IF  Mach_Control.U.WJ_iMode=3 AND arrAxisCtrl[AxiseNo.AxisName.TailCurlLine].Status.Homed 
AND arrAxisCtrl[AxiseNo.AxisName.TailCurlWhirling].Cmd.arrbRealPoint[1] 
AND arrAxisCtrl[AxiseNo.AxisName.LCurlingneedleLine].Status.fActPos<=arrAxisPar[AxiseNo.AxisName.LCurlingneedleLine].arrTargetPoint[1] +1
AND arrAxisCtrl[AxiseNo.AxisName.LCurlingneedleLine].Status.Homed  
AND arrAxisCtrl[AxiseNo.AxisName.SCurlingneedleLine].Status.fActPos <=arrAxisPar[AxiseNo.AxisName.SCurlingneedleLine] .arrTargetPoint[1] +1
AND arrAxisCtrl[AxiseNo.AxisName.SCurlingneedleLine].Status.Homed 
OR Mach_Control.WJ_b.AxisConditionEN THEN
	arrAxisCtrl[AxiseNo.AxisName.TailCurlLine].Cmd.GoPoint_Condition[10]:=TRUE;
ELSE
	arrAxisCtrl[AxiseNo.AxisName.TailCurlLine].Cmd.GoPoint_Condition[10]:=FALSE;	
END_IF

IF  Mach_Control.U.WJ_iMode=3 AND   arrAxisCtrl[AxiseNo.AxisName.TailCurlLine].Status.Homed  AND   arrAxisCtrl[AxiseNo.AxisName.TailCurlWhirling].Cmd.arrbRealPoint[1] AND
	(arrAxisCtrl[AxiseNo.AxisName.LCurlingneedleLine].Status.fActPos<=arrAxisPar[AxiseNo.AxisName.LCurlingneedleLine].arrTargetPoint[1]+1 AND arrAxisCtrl[AxiseNo.AxisName.LCurlingneedleLine].Status.Homed  AND
	arrAxisCtrl[AxiseNo.AxisName.SCurlingneedleLine].Status.fActPos <=arrAxisPar[AxiseNo.AxisName.SCurlingneedleLine] .arrTargetPoint[1]+1 AND arrAxisCtrl[AxiseNo.AxisName.SCurlingneedleLine].Status.Homed  AND
	arrAxisCtrl[AxiseNo.AxisName.TailCurlSEPTAUpDown].Cmd.arrbRealPoint[1] ) AND  arrCyCtrl[arrCyNo.CylinderName.PoleSplintCy_D].Status.OFFState AND
    arrAxisCtrl[AxiseNo.AxisName.TailCurlSEPTALine].Cmd.arrbRealPoint[1] OR Mach_Control.WJ_b.AxisConditionEN THEN
    arrAxisCtrl[AxiseNo.AxisName.TailCurlLine].Cmd.GoPoint_Condition[11]:=TRUE;
ELSE
	arrAxisCtrl[AxiseNo.AxisName.TailCurlLine].Cmd.GoPoint_Condition[11]:=FALSE;	
END_IF


//尾卷夹电芯伸缩
IF  Mach_Control.U.WJ_iMode=3  
OR Mach_Control.WJ_b.AxisConditionEN THEN
	arrAxisCtrl[AxiseNo.AxisName.TailCurlRetracting].Cmd.Home_Condition:=TRUE;
ELSE
	arrAxisCtrl[AxiseNo.AxisName.TailCurlRetracting].Cmd.Home_Condition:=FALSE;	
END_IF

IF  Mach_Control.U.WJ_iMode=3 AND arrAxisCtrl[AxiseNo.AxisName.TailCurlRetracting].Status.Homed 
OR Mach_Control.WJ_b.AxisConditionEN THEN
	arrAxisCtrl[AxiseNo.AxisName.TailCurlRetracting].Cmd.GoPoint_Condition[1]:=TRUE;
ELSE
	arrAxisCtrl[AxiseNo.AxisName.TailCurlRetracting].Cmd.GoPoint_Condition[1]:=FALSE;	
END_IF

IF  Mach_Control.U.WJ_iMode=3 AND arrAxisCtrl[AxiseNo.AxisName.TailCurlRetracting].Status.Homed 
OR Mach_Control.WJ_b.AxisConditionEN THEN
	arrAxisCtrl[AxiseNo.AxisName.TailCurlRetracting].Cmd.GoPoint_Condition[2]:=TRUE;
ELSE
	arrAxisCtrl[AxiseNo.AxisName.TailCurlRetracting].Cmd.GoPoint_Condition[2]:=FALSE;	
END_IF

IF  Mach_Control.U.WJ_iMode=3 AND arrAxisCtrl[AxiseNo.AxisName.TailCurlRetracting].Status.Homed 
OR Mach_Control.WJ_b.AxisConditionEN THEN
	arrAxisCtrl[AxiseNo.AxisName.TailCurlRetracting].Cmd.GoPoint_Condition[3]:=TRUE;
ELSE
	arrAxisCtrl[AxiseNo.AxisName.TailCurlRetracting].Cmd.GoPoint_Condition[3]:=FALSE;	
END_IF


//尾卷夹膜平移
IF  Mach_Control.U.WJ_iMode=3 AND
    arrAxisCtrl[AxiseNo.AxisName.CaDTCarryingUpDown].Status.fActPos<=arrAxisPar[AxiseNo.AxisName.CaDTCarryingUpDown].arrTargetPoint[5]+1 AND arrAxisCtrl[AxiseNo.AxisName.CaDTCarryingUpDown].Status.Homed AND
	arrAxisCtrl[AxiseNo.AxisName.CaDTCarryingLine].Status.Homed AND arrAxisCtrl[AxiseNo.AxisName.CaDTCarryingLine].Cmd.arrbRealPoint[1] 	 THEN
       arrAxisCtrl[AxiseNo.AxisName.TailCurlSEPTALine].Cmd.JogP_Condition:=TRUE;
ELSE 
	   arrAxisCtrl[AxiseNo.AxisName.TailCurlSEPTALine].Cmd.JogP_Condition:=FALSE;
END_IF 
 
IF  Mach_Control.U.WJ_iMode=3 AND
	arrAxisCtrl[AxiseNo.AxisName.TailCurlLine].Status.fActPos<=arrAxisPar[AxiseNo.AxisName.TailCurlLine].arrTargetPoint[4]+1 AND arrAxisCtrl[AxiseNo.AxisName.TailCurlLine].Status.Homed 
    OR Mach_Control.WJ_b.AxisConditionEN THEN
		arrAxisCtrl[AxiseNo.AxisName.TailCurlSEPTALine].Cmd.Home_Condition:=TRUE;
		arrAxisCtrl[AxiseNo.AxisName.TailCurlSEPTALine].Cmd.GoPoint_Condition[1]:=TRUE;
		//TailCurlSEPTALineGoargee:=TRUE;
ELSE
		arrAxisCtrl[AxiseNo.AxisName.TailCurlSEPTALine].Cmd.Home_Condition:=FALSE;	
		arrAxisCtrl[AxiseNo.AxisName.TailCurlSEPTALine].Cmd.GoPoint_Condition[1]:=FALSE;
		//TailCurlSEPTALineGoargee:=FALSE;
END_IF

IF  Mach_Control.U.WJ_iMode=3 AND
	arrAxisCtrl[AxiseNo.AxisName.CaDTCarryingUpDown].Status.fActPos<=arrAxisPar[AxiseNo.AxisName.CaDTCarryingUpDown].arrTargetPoint[5]+1 AND arrAxisCtrl[AxiseNo.AxisName.CaDTCarryingUpDown].Status.Homed AND
	arrAxisCtrl[AxiseNo.AxisName.CaDTCarryingLine].Status.Homed AND arrAxisCtrl[AxiseNo.AxisName.CaDTCarryingLine].Cmd.arrbRealPoint[1] 
OR Mach_Control.WJ_b.AxisConditionEN THEN
		arrAxisCtrl[AxiseNo.AxisName.TailCurlSEPTALine].Cmd.Home_Condition:=TRUE;

		arrAxisCtrl[AxiseNo.AxisName.TailCurlSEPTALine].Cmd.GoPoint_Condition[2]:=TRUE;
		//TailCurlSEPTALineGoargee:=TRUE;
ELSE
		arrAxisCtrl[AxiseNo.AxisName.TailCurlSEPTALine].Cmd.Home_Condition:=FALSE;	

		arrAxisCtrl[AxiseNo.AxisName.TailCurlSEPTALine].Cmd.GoPoint_Condition[2]:=FALSE;
		//TailCurlSEPTALineGoargee:=FALSE;
END_IF

(*
IF  Mach_Control.U.DT_iMode=3 AND arrAxisCtrl[AxiseNo.AxisName.CaCarryingLine2].Cmd.arrbRealPoint[1] 
AND (arrAxisCtrl[AxiseNo.AxisName.TailCurlLine].Cmd.arrbRealPoint[5] OR arrAxisCtrl[AxiseNo.AxisName.TailCurlLine].Cmd.arrbRealPoint[6] OR arrAxisCtrl[AxiseNo.AxisName.TailCurlLine].Cmd.arrbRealPoint[1])
AND (arrAxisCtrl[AxiseNo.AxisName.TailCurlWhirling].Cmd.arrbRealPoint[1] OR  arrAxisCtrl[AxiseNo.AxisName.TailCurlWhirling].Cmd.arrbRealPoint[2]) THEN
	arrAxisCtrl[AxiseNo.AxisName.TailCurlSEPTALine].Cmd.GoPoint_Condition[1]:=TRUE;
ELSE
	arrAxisCtrl[AxiseNo.AxisName.TailCurlSEPTALine].Cmd.GoPoint_Condition[1]:=FALSE;	
END_IF

IF  Mach_Control.U.DT_iMode=3 AND arrAxisCtrl[AxiseNo.AxisName.CaCarryingLine2].Cmd.arrbRealPoint[1] 
AND (arrAxisCtrl[AxiseNo.AxisName.TailCurlLine].Cmd.arrbRealPoint[5] OR arrAxisCtrl[AxiseNo.AxisName.TailCurlLine].Cmd.arrbRealPoint[6] OR arrAxisCtrl[AxiseNo.AxisName.TailCurlLine].Cmd.arrbRealPoint[1])
AND (arrAxisCtrl[AxiseNo.AxisName.TailCurlWhirling].Cmd.arrbRealPoint[1] OR  arrAxisCtrl[AxiseNo.AxisName.TailCurlWhirling].Cmd.arrbRealPoint[2]) THEN
	arrAxisCtrl[AxiseNo.AxisName.TailCurlSEPTALine].Cmd.GoPoint_Condition[2]:=TRUE;
ELSE
	arrAxisCtrl[AxiseNo.AxisName.TailCurlSEPTALine].Cmd.GoPoint_Condition[2]:=FALSE;	
END_IF
*)

//尾卷夹膜升降
IF  Mach_Control.U.WJ_iMode=3 AND
	 arrAxisCtrl[AxiseNo.AxisName.TailCurlLine].Status.fSetPos<=arrAxisPar[AxiseNo.AxisName.TailCurlLine].arrTargetPoint[4] AND arrAxisCtrl[AxiseNo.AxisName.TailCurlLine].Status.Homed    
OR Mach_Control.WJ_b.AxisConditionEN THEN
		arrAxisCtrl[AxiseNo.AxisName.TailCurlSEPTAUpDown].Cmd.Home_Condition:=TRUE;
ELSE
	arrAxisCtrl[AxiseNo.AxisName.TailCurlSEPTAUpDown].Cmd.Home_Condition:=FALSE;	
END_IF

IF  Mach_Control.U.WJ_iMode=3 AND arrAxisCtrl[AxiseNo.AxisName.TailCurlSEPTAUpDown].Status.Homed 
AND NOT arrAxisCtrl[AxiseNo.AxisName.TailCurlLine].Cmd.arrbRealPoint[11] OR Mach_Control.WJ_b.AxisConditionEN THEN
	arrAxisCtrl[AxiseNo.AxisName.TailCurlSEPTAUpDown].Cmd.GoPoint_Condition[1]:=TRUE;
ELSE
	arrAxisCtrl[AxiseNo.AxisName.TailCurlSEPTAUpDown].Cmd.GoPoint_Condition[1]:=FALSE;	
END_IF

IF  Mach_Control.U.WJ_iMode=3 AND arrAxisCtrl[AxiseNo.AxisName.TailCurlSEPTAUpDown].Status.Homed  
AND arrAxisCtrl[AxiseNo.AxisName.TailCurlLine].Status.fActPos <=  arrAxisPar[AxiseNo.AxisName.TailCurlLine].arrTargetPoint[4]  
AND NOT arrAxisCtrl[AxiseNo.AxisName.TailCurlLine].Cmd.arrbRealPoint[11] OR Mach_Control.WJ_b.AxisConditionEN THEN
	arrAxisCtrl[AxiseNo.AxisName.TailCurlSEPTAUpDown].Cmd.GoPoint_Condition[2]:=TRUE;
ELSE
	arrAxisCtrl[AxiseNo.AxisName.TailCurlSEPTAUpDown].Cmd.GoPoint_Condition[2]:=FALSE;	
END_IF

//尾卷夹电芯升降
IF  Mach_Control.U.WJ_iMode=3 AND  arrAxisCtrl[AxiseNo.AxisName.TailCurlRetracting].Cmd.arrbRealPoint[1] 
OR Mach_Control.WJ_b.AxisConditionEN THEN
	arrAxisCtrl[AxiseNo.AxisName.TailCurlUpDown].Cmd.Home_Condition:=TRUE;
ELSE
	arrAxisCtrl[AxiseNo.AxisName.TailCurlUpDown].Cmd.Home_Condition:=FALSE;	
END_IF

IF  Mach_Control.U.WJ_iMode=3 
AND arrAxisCtrl[AxiseNo.AxisName.TailCurlSEPTAUpDown].Status.Homed  
AND  arrAxisCtrl[AxiseNo.AxisName.TailCurlRetracting].Cmd.arrbRealPoint[1] 
AND NOT arrAxisCtrl[AxiseNo.AxisName.TailCurlLine].Cmd.arrbRealPoint[6]
OR Mach_Control.WJ_b.AxisConditionEN THEN
	arrAxisCtrl[AxiseNo.AxisName.TailCurlUpDown].Cmd.GoPoint_Condition[1]:=TRUE;
ELSE
	arrAxisCtrl[AxiseNo.AxisName.TailCurlUpDown].Cmd.GoPoint_Condition[1]:=FALSE;	
END_IF
////////////////////////////////////////////
IF  Mach_Control.U.WJ_iMode=3 
AND arrAxisCtrl[AxiseNo.AxisName.TailCurlSEPTAUpDown].Status.Homed  
AND arrAxisCtrl[AxiseNo.AxisName.TailCurlWhirling].Cmd.arrbRealPoint[1]
AND arrAxisCtrl[AxiseNo.AxisName.TailCurlRetracting].Cmd.arrbRealPoint[1] 
AND  arrAxisCtrl[AxiseNo.AxisName.TailCurlLine].Status.fActPos <=  arrAxisPar[AxiseNo.AxisName.TailCurlLine].arrTargetPoint[4]  
OR Mach_Control.WJ_b.AxisConditionEN THEN
	arrAxisCtrl[AxiseNo.AxisName.TailCurlUpDown].Cmd.GoPoint_Condition[2]:=TRUE;
ELSE
	arrAxisCtrl[AxiseNo.AxisName.TailCurlUpDown].Cmd.GoPoint_Condition[2]:=FALSE;	
END_IF

IF  Mach_Control.U.WJ_iMode=3 
AND arrAxisCtrl[AxiseNo.AxisName.TailCurlSEPTAUpDown].Status.Homed 
AND arrAxisCtrl[AxiseNo.AxisName.TailCurlRetracting].Cmd.arrbRealPoint[1]
AND NOT arrAxisCtrl[AxiseNo.AxisName.TailCurlLine].Cmd.arrbRealPoint[11] 
OR Mach_Control.WJ_b.AxisConditionEN THEN
	arrAxisCtrl[AxiseNo.AxisName.TailCurlUpDown].Cmd.GoPoint_Condition[3]:=TRUE;

ELSE
	arrAxisCtrl[AxiseNo.AxisName.TailCurlUpDown].Cmd.GoPoint_Condition[3]:=FALSE;	
END_IF

IF  Mach_Control.U.WJ_iMode=3 
AND arrAxisCtrl[AxiseNo.AxisName.TailCurlSEPTAUpDown].Status.Homed
AND arrAxisCtrl[AxiseNo.AxisName.TailCurlWhirling].Cmd.arrbRealPoint[2]  
AND arrAxisCtrl[AxiseNo.AxisName.TailCurlRetracting].Cmd.arrbRealPoint[1]
AND NOT arrAxisCtrl[AxiseNo.AxisName.TailCurlLine].Cmd.arrbRealPoint[11] 
OR Mach_Control.WJ_b.AxisConditionEN THEN
	arrAxisCtrl[AxiseNo.AxisName.TailCurlUpDown].Cmd.GoPoint_Condition[4]:=TRUE;
ELSE
	arrAxisCtrl[AxiseNo.AxisName.TailCurlUpDown].Cmd.GoPoint_Condition[4]:=FALSE;	
END_IF
///////////////////////////////////////////
//尾卷夹电芯旋转 
IF  Mach_Control.U.WJ_iMode=3 AND  arrAxisCtrl[AxiseNo.AxisName.TailCurlRetracting].Cmd.arrbRealPoint[1] AND arrAxisCtrl[AxiseNo.AxisName.TailCurlLine].Cmd.arrbRealPoint[1] AND
   arrAxisCtrl[AxiseNo.AxisName.TailCurlRetracting].Status.Homed AND arrAxisCtrl[AxiseNo.AxisName.TailCurlLine].Status.Homed 	
OR Mach_Control.WJ_b.AxisConditionEN THEN
	arrAxisCtrl[AxiseNo.AxisName.TailCurlWhirling].Cmd.Home_Condition:=TRUE;
ELSE
	arrAxisCtrl[AxiseNo.AxisName.TailCurlWhirling].Cmd.Home_Condition:=FALSE;	
END_IF

IF  Mach_Control.U.WJ_iMode=3 AND arrAxis[AxiseNo.AxisName.TailCurlWhirling].Status.Homed  AND  arrAxisCtrl[AxiseNo.AxisName.TailCurlRetracting].Cmd.arrbRealPoint[1] 
AND arrAxisCtrl[AxiseNo.AxisName.TailCurlUpDown].Cmd.arrbRealPoint[3] AND arrAxisCtrl[AxiseNo.AxisName.TailCurlLine].Cmd.arrbRealPoint[1] 
OR Mach_Control.WJ_b.AxisConditionEN THEN
	arrAxisCtrl[AxiseNo.AxisName.TailCurlWhirling].Cmd.GoPoint_Condition[1]:=TRUE;
ELSE
	arrAxisCtrl[AxiseNo.AxisName.TailCurlWhirling].Cmd.GoPoint_Condition[1]:=FALSE;	
END_IF

IF  Mach_Control.U.WJ_iMode=3 AND arrAxis[AxiseNo.AxisName.TailCurlWhirling].Status.Homed  AND  arrAxisCtrl[AxiseNo.AxisName.TailCurlRetracting].Cmd.arrbRealPoint[1] 
AND arrAxisCtrl[AxiseNo.AxisName.TailCurlUpDown].Cmd.arrbRealPoint[3] AND arrAxisCtrl[AxiseNo.AxisName.TailCurlLine].Cmd.arrbRealPoint[1] 
OR Mach_Control.WJ_b.AxisConditionEN THEN
	arrAxisCtrl[AxiseNo.AxisName.TailCurlWhirling].Cmd.GoPoint_Condition[2]:=TRUE;
ELSE
	arrAxisCtrl[AxiseNo.AxisName.TailCurlWhirling].Cmd.GoPoint_Condition[2]:=FALSE;	
END_IF

//尾卷长卷针平移
IF  Mach_Control.U.WJ_iMode=3 
OR Mach_Control.WJ_b.AxisConditionEN THEN
	arrAxisCtrl[AxiseNo.AxisName.LCurlingneedleLine].Cmd.Home_Condition:=TRUE;
ELSE
	arrAxisCtrl[AxiseNo.AxisName.LCurlingneedleLine].Cmd.Home_Condition:=FALSE;	
END_IF

IF  Mach_Control.U.WJ_iMode=3 AND arrAxisCtrl[AxiseNo.AxisName.LCurlingneedleLine].Status.Homed AND arrCyCtrl[arrCyNo.CylinderName.CurlingSplintCy_L].Status.OFFState
OR Mach_Control.WJ_b.AxisConditionEN THEN
	arrAxisCtrl[AxiseNo.AxisName.LCurlingneedleLine].Cmd.GoPoint_Condition[1]:=TRUE;
ELSE
	arrAxisCtrl[AxiseNo.AxisName.LCurlingneedleLine].Cmd.GoPoint_Condition[1]:=FALSE;	
END_IF

IF  Mach_Control.U.WJ_iMode=3 AND arrAxisCtrl[AxiseNo.AxisName.LCurlingneedleLine].Status.Homed AND arrCyCtrl[arrCyNo.CylinderName.CurlingSplintCy_L].Status.OFFState
     AND  arrAxisCtrl[AxiseNo.AxisName.TailCurlLine].Cmd.arrbRealPoint[4]   OR Mach_Control.WJ_b.AxisConditionEN THEN
	arrAxisCtrl[AxiseNo.AxisName.LCurlingneedleLine].Cmd.GoPoint_Condition[2]:=TRUE;
ELSE
	arrAxisCtrl[AxiseNo.AxisName.LCurlingneedleLine].Cmd.GoPoint_Condition[2]:=FALSE;	
END_IF


//尾卷短卷针平移
IF  (Mach_Control.U.WJ_iMode=3  AND arrAxisCtrl[AxiseNo.AxisName.SCurlingneedleWhirling].Io.biHomeSwitch)
OR Mach_Control.WJ_b.AxisConditionEN   THEN
	arrAxisCtrl[AxiseNo.AxisName.SCurlingneedleLine].Cmd.Home_Condition:=TRUE;
ELSE
	arrAxisCtrl[AxiseNo.AxisName.SCurlingneedleLine].Cmd.Home_Condition:=FALSE;	
END_IF

IF  Mach_Control.U.WJ_iMode=3 AND arrAxisCtrl[AxiseNo.AxisName.SCurlingneedleLine].Status.Homed  AND arrCyCtrl[arrCyNo.CylinderName.CurlingSplintCy_S].Status.OFFState
OR Mach_Control.WJ_b.AxisConditionEN THEN
	arrAxisCtrl[AxiseNo.AxisName.SCurlingneedleLine].Cmd.GoPoint_Condition[1]:=TRUE;
ELSE
	arrAxisCtrl[AxiseNo.AxisName.SCurlingneedleLine].Cmd.GoPoint_Condition[1]:=FALSE;	
END_IF

IF  Mach_Control.U.WJ_iMode=3 AND arrAxisCtrl[AxiseNo.AxisName.SCurlingneedleLine].Status.Homed  AND arrCyCtrl[arrCyNo.CylinderName.CurlingSplintCy_S].Status.OFFState
    AND  arrCyCtrl[arrCyNo.ElectValveName.WJShortvacuum].Io.DOStatus1 AND  arrAxisCtrl[AxiseNo.AxisName.TailCurlLine].Cmd.arrbRealPoint[4]    OR Mach_Control.WJ_b.AxisConditionEN THEN
	arrAxisCtrl[AxiseNo.AxisName.SCurlingneedleLine].Cmd.GoPoint_Condition[2]:=TRUE;
ELSE
	arrAxisCtrl[AxiseNo.AxisName.SCurlingneedleLine].Cmd.GoPoint_Condition[2]:=FALSE;	
END_IF

//尾卷长卷针旋转
IF  Mach_Control.U.WJ_iMode=3 AND arrAxisCtrl[AxiseNo.AxisName.LCurlingneedleLine].Status.fSetPos<=arrAxisPar[AxiseNo.AxisName.LCurlingneedleLine].arrTargetPoint[1]  
OR Mach_Control.WJ_b.AxisConditionEN THEN
	arrAxisCtrl[AxiseNo.AxisName.LCurlingneedleWhirling].Cmd.Home_Condition:=TRUE;
ELSE
	arrAxisCtrl[AxiseNo.AxisName.LCurlingneedleWhirling].Cmd.Home_Condition:=FALSE;	
END_IF

IF  Mach_Control.U.WJ_iMode=3 AND arrAxisCtrl[AxiseNo.AxisName.LCurlingneedleWhirling].Status.Homed 
AND arrAxisCtrl[AxiseNo.AxisName.LCurlingneedleLine].Cmd.arrbRealPoint[1]  
OR Mach_Control.WJ_b.AxisConditionEN THEN
	arrAxisCtrl[AxiseNo.AxisName.LCurlingneedleWhirling].Cmd.GoPoint_Condition[1]:=TRUE;
ELSE
	arrAxisCtrl[AxiseNo.AxisName.LCurlingneedleWhirling].Cmd.GoPoint_Condition[1]:=FALSE;	
END_IF

//尾卷短卷针旋转
IF  Mach_Control.U.WJ_iMode=3 AND arrAxisCtrl[AxiseNo.AxisName.SCurlingneedleLine].Status.fSetPos<=arrAxisPar[AxiseNo.AxisName.SCurlingneedleLine].arrTargetPoint[1]  
OR Mach_Control.WJ_b.AxisConditionEN THEN
	arrAxisCtrl[AxiseNo.AxisName.SCurlingneedleWhirling].Cmd.Home_Condition:=TRUE;
ELSE
	arrAxisCtrl[AxiseNo.AxisName.SCurlingneedleWhirling].Cmd.Home_Condition:=FALSE;	
END_IF

IF  Mach_Control.U.WJ_iMode=3 AND arrAxisCtrl[AxiseNo.AxisName.SCurlingneedleWhirling].Status.Homed 
AND arrAxisCtrl[AxiseNo.AxisName.SCurlingneedleLine].Cmd.arrbRealPoint[1]  
OR Mach_Control.WJ_b.AxisConditionEN THEN
	arrAxisCtrl[AxiseNo.AxisName.SCurlingneedleWhirling].Cmd.GoPoint_Condition[1]:=TRUE;
ELSE
	arrAxisCtrl[AxiseNo.AxisName.SCurlingneedleWhirling].Cmd.GoPoint_Condition[1]:=FALSE;	
END_IF
END_ACTION

ACTION TailCurl_Gohome:
Tailcurl_GohomeOverTon(IN:= , PT:=T#90S , Q=> , ET=> );//叠台回原点超时报警延时

//判断回原点的状态
IF arrAxisCtrl[AxiseNo.AxisName.SCurlingneedleLine].Status.Homed AND arrAxisCtrl[AxiseNo.AxisName.LCurlingneedleLine].Status.Homed AND 
	arrAxisCtrl[AxiseNo.AxisName.LCurlingneedleWhirling].Status.Homed  AND arrAxisCtrl[AxiseNo.AxisName.SCurlingneedleWhirling].Status.Homed AND 
	arrAxisCtrl[AxiseNo.AxisName.TailCurlLine].Status.Homed AND arrAxisCtrl[AxiseNo.AxisName.TailCurlRetracting].Status.Homed AND 
	arrAxisCtrl[AxiseNo.AxisName.TailCurlUpDown].Status.Homed AND arrAxisCtrl[AxiseNo.AxisName.TailCurlSEPTAUpDown].Status.Homed AND 
	arrAxis[AxiseNo.AxisName.TailCurlSEPTALine].Status.Homed AND arrAxis[AxiseNo.AxisName.TailCurlWhirling].Status.Homed AND WZIniti_Done THEN
		Mach_Control.WJ_b.WZIniti_Done:=TRUE;//初始化完成	
ELSE
		Mach_Control.WJ_b.WZIniti_Done:=FALSE;//初始化完成	
END_IF

IF Mach_Control.U.WJ_iMode=3 THEN//在手动状态下
	IF  Tailcurl_Gohoming THEN
			IF 	NOT Tailcurl_GohomeOverTon.Q THEN
				    Tailcurl_GohomeOverTon.IN:=TRUE;
			ELSE
				IF 	Tailcurl_GohomeOverTon.Q THEN
					Tailcurl_Gohoming:=FALSE;
					TailCurlStep1:=0;
				     Mach_Control.WJ_b.Error[19]:=TRUE;//尾卷回原点超时报警
				     Tailcurl_GohomeOverTon.IN:=FALSE;
				END_IF	 
					 
			END_IF
	
	ELSE
			Tailcurl_GohomeOverTon.IN:=FALSE;
	END_IF
	
	IF r_TailCurl_init.Q THEN
		Tailcurl_GohomeDone:=FALSE;//尾卷回原点完成
		Tailcurl_Gohoming:=FALSE;//尾卷回原点中
		TailCurlStep1:=0;
		Mach_Control.WJ_b.WZIniti_Done:=FALSE;//负极取片回原点完成
		WZIniti_Done:=FALSE;//负极取片回原点完成
	END_IF	

	//尾卷贴胶初始化
	r_TailCurl_init(CLK:=Mach_Control.WJ_b.WZIniti_Hbtn , Q=> );
	f_TailCurl_init(CLK:=Mach_Control.WJ_b.WZIniti_Hbtn   , Q=> );
	tTailCurlTON(IN:= , PT:=T#0.5S , Q=> , ET=> );
	CASE TailCurlStep1 OF
	0://启动尾卷贴胶初始化，气缸复位
		IF f_TailCurl_init.Q THEN	
			Tailcurl_GohomeDone:=FALSE;//尾卷回原点完成
		    Tailcurl_Gohoming:=TRUE;//尾卷回原点中
			TailCurlStep1:=1;
		END_IF
	1://回原点完成复位
			WZIniti_Done:=FALSE;//初始化完成	
			TailCurlStep3 :=0;
			TailCurlStep4:=0;
			TailCurlStep5:=0;
			TailCurlStep6:=0;
			
			arrAxisCtrl[AxiseNo.AxisName.TailCurlSEPTALine].Cmd.fOverride:=100;
			arrAxisCtrl[AxiseNo.AxisName.TailCurlRetracting].Cmd.fOverride:=100;
			arrAxisCtrl[AxiseNo.AxisName.TailCurlLine].Cmd.fOverride:=100;
						
			tailCult_GearInMultiMaster.Enable:=FALSE;
			tailCurlGearInEnable:=FALSE;
			tailCurlGearInEnable1:=FALSE;
			tailRetGearInEnable:=FALSE;//夹电芯平移与夹电芯伸缩电子齿轮
			CurlingneedleLineEnable:=FALSE;
			tailCult_GearInMultiMaster.Enable:=FALSE;
			
			 Mach_Control.DT_b.OffloadDone:=FALSE;
			 Mach_Control.WJ_b.TailCurlDone	:=FALSE;
			 //Mach_Control.DT_b.OffloadRequest:=FALSE;//复位电芯下料请求	
			 Mach_Control.WJ_b.TailCultOffloading:=FALSE;
			CellMemory[Mach_Control.WJ_b.WJ_Memory].Cell:=FALSE;	
			TailCurlStart:=FALSE;//复位尾卷启动
			Mach_Control.WJ_b.TailCurlDone	:=FALSE;	//尾卷完成
			arrAxisCtrl[AxiseNo.VirAxisName.VirTailCurl].Cmd.bMoveAbs:=FALSE;//主轴启动
			CurlingneedleLineEnable:=FALSE;//长、短卷针平移电子齿轮耦合启动
			tailCurlGearInEnable:=FALSE;//电子齿轮耦合		
			tTailCurlTON.IN:=FALSE;
			arrAxisCtrl[AxiseNo.AxisName.TailCurlSEPTALine].Cmd.bDynamitcsParSel:=1;
			fbCamInEndWindX.bGearOutMode:=FALSE;//夹膜平移轴凸轮耦合
			IF NOT WZIniti_Done AND arrAxisCtrl[AxiseNo.AxisName.TailCurlSEPTALine].Cmd.bDynamitcsParSel=1 THEN
				TailCurlStep1:=10;
			END_IF
	10://气缸复位，尾卷状态复位
			IF  NOT 	tTailCurlTON.Q THEN	
					tTailCurlTON.IN:=TRUE;
					//arrCyCtrl[arrCyNo.CylinderName.CurlingSplintCy_S_1].Cmd.bON:=TRUE;//尾卷短卷针泄压关闭
					arrCyCtrl[arrCyNo.CylinderName.CurlingSplintCy_L].Cmd.bOFF:=TRUE;//尾卷长卷针张开
					arrCyCtrl[arrCyNo.CylinderName.CurlingSplintCy_S].Cmd.bOFF:=TRUE;//尾卷短卷针张开	
					arrCyCtrl[arrCyNo.ElectValveName.WJShortvacuum].Cmd.bON:=TRUE;//短卷针张开真空开
					arrCyCtrl[arrCyNo.CylinderName.PoleHotCutterCy].Cmd.bOFF:=TRUE;//隔膜热切升降气缸收回
					arrCyCtrl[arrCyNo.CylinderName.PoleSplintCy_D].Cmd.bOFF:=TRUE;//隔膜隔膜下夹板气缸收回
					arrCyCtrl[arrCyNo.CylinderName.TailCurlUpdownCy].Cmd.bOFF:=TRUE;//尾卷压轮升降气缸收回
					arrCyCtrl[arrCyNo.CylinderName.TailCurlSplintCy].Cmd.bOFF:=TRUE;//尾卷取料夹爪气缸张开	
			ELSE
					IF arrCyCtrl[arrCyNo.CylinderName.PoleHotCutterCy].Io.DIOFFSwitch AND arrCyCtrl[arrCyNo.CylinderName.PoleSplintCy_D].Io.DIOFFSwitch AND 
					   arrCyCtrl[arrCyNo.CylinderName.TailCurlUpdownCy].Io.DIOFFSwitch AND arrCyCtrl[arrCyNo.CylinderName.TailCurlSplintCy].Io.DIOFFSwitch THEN
					   tTailCurlTON.IN:=FALSE;
					   TailCurlStep1:=20;
					END_IF	
			END_IF	
	20:
			fbCamInEndWindX.bCamInExecute:=FALSE;//夹膜平移凸轮耦合
			fbCamInEndWindY.bCamInExecute:=FALSE;//夹膜升降凸轮耦合
			tailCurl1_GearIn.Execute:=FALSE;//短卷针齿轮耦合
			tailCurl2_GearIn.Execute:=FALSE;//长卷针齿轮耦合
			IF NOT fbCamInEndWindX.bCamInExecute AND NOT fbCamInEndWindY.bCamInExecute AND 
				NOT tailCurl1_GearIn.Execute AND NOT tailCurl2_GearIn.Execute THEN
				TailCurlStep1:=21;
			END_IF
	21://解除凸轮耦合
			arrCyCtrl[arrCyNo.CylinderName.TailCurlLineCy].Cmd.bOFF:=TRUE;//尾卷压轮平移气缸收回
			arrAxisCtrl[AxiseNo.AxisName.SCurlingneedleWhirling].Cmd.bGearOut:=TRUE;//尾卷短卷针旋转轴解耦
			arrAxisCtrl[AxiseNo.AxisName.LCurlingneedleWhirling].Cmd.bGearOut:=TRUE;//尾卷长卷针旋转轴解耦
			arrAxisCtrl[AxiseNo.AxisName.TailCurlLine].Cmd.bGearOut:=TRUE;//尾卷夹电芯平移轴解耦
			arrAxisCtrl[AxiseNo.AxisName.TailCurlSEPTALine].Cmd.bGearOut:=TRUE;//尾卷夹膜平移轴解耦 
			arrAxisCtrl[AxiseNo.AxisName.TailCurlSEPTAUpDown].Cmd.bGearOut:=TRUE;//尾卷夹膜升降轴解耦 
			IF NOT arrAxisCtrl[AxiseNo.AxisName.SCurlingneedleWhirling].Status.Coupled AND  NOT arrAxisCtrl[AxiseNo.AxisName.LCurlingneedleWhirling].Status.Coupled AND 
				NOT arrAxisCtrl[AxiseNo.AxisName.TailCurlLine].Status.Coupled AND NOT arrAxisCtrl[AxiseNo.AxisName.TailCurlSEPTALine].Status.Coupled AND 
				NOT arrAxisCtrl[AxiseNo.AxisName.TailCurlSEPTAUpDown].Status.Coupled THEN
				TailCurlStep1:=25;
			END_IF

	 25:
		 IF NOT arrAxisCtrl[AxiseNo.AxisName.SCurlingneedleWhirling].Io.biHomeSwitch  THEN
			  Mach_Control.WJ_b.Error[20]:=TRUE;//尾卷短卷针神伸缩回原点时,短卷针旋转原点传感器未亮报警
			  TailCurlStep1:=0;
		  ELSE 	 
			 TailCurlStep1:=30;
		 END_IF			
			

    30://尾卷长卷针伸缩轴回原点、尾卷短卷针伸缩轴回原点	
						IF NOT tTailCurlTON.Q THEN
								arrAxisCtrl[AxiseNo.AxisName.SCurlingneedleLine].Cmd.bHome:=TRUE;//尾卷短卷针平移回原点
								arrAxisCtrl[AxiseNo.AxisName.LCurlingneedleLine].Cmd.bHome:=TRUE;//尾卷长卷针平移回原点
								tTailCurlTON.IN:=TRUE;
						ELSE
								IF arrAxisCtrl[AxiseNo.AxisName.SCurlingneedleLine].Status.Homed AND arrAxisCtrl[AxiseNo.AxisName.SCurlingneedleLine].Status.NoMoving  AND
									 arrAxisCtrl[AxiseNo.AxisName.LCurlingneedleLine].Status.Homed AND arrAxisCtrl[AxiseNo.AxisName.LCurlingneedleLine].Status.NoMoving THEN
										arrAxisCtrl[AxiseNo.AxisName.SCurlingneedleLine].Cmd.bHome:=FALSE;//尾卷短卷针平移回原点
										arrAxisCtrl[AxiseNo.AxisName.LCurlingneedleLine].Cmd.bHome:=FALSE;//尾卷长卷针平移回原点
										tTailCurlTON.IN:=FALSE;
										TailCurlStep1:=35; 
								END_IF
						END_IF
			
		35:
						IF 	arrAxisCtrl[AxiseNo.AxisName.LCurlingneedleLine].Status.Homed AND arrAxisCtrl[AxiseNo.AxisName.LCurlingneedleLine].Status.NoMoving THEN
							IF arrAxisCtrl[AxiseNo.AxisName.LCurlingneedleLine].Cmd.arrbRealPoint[1] THEN
								arrAxisCtrl[AxiseNo.AxisName.LCurlingneedleLine].Cmd.iGoSetPos:=0;
							ELSE
								arrAxisCtrl[AxiseNo.AxisName.LCurlingneedleLine].Cmd.iGoSetPos:=1;//尾卷长卷针平移至初始位
							END_IF
						END_IF	
						IF 	arrAxisCtrl[AxiseNo.AxisName.SCurlingneedleLine].Status.Homed AND arrAxisCtrl[AxiseNo.AxisName.SCurlingneedleLine].Status.NoMoving THEN
							IF arrAxisCtrl[AxiseNo.AxisName.SCurlingneedleLine].Cmd.arrbRealPoint[1] THEN
								arrAxisCtrl[AxiseNo.AxisName.SCurlingneedleLine].Cmd.iGoSetPos:=0;
							ELSE
								arrAxisCtrl[AxiseNo.AxisName.SCurlingneedleLine].Cmd.iGoSetPos:=1;//尾卷短卷针平移至初始位
							END_IF
						END_IF		
							IF 	arrAxisCtrl[AxiseNo.AxisName.LCurlingneedleLine].Cmd.arrbRealPoint[1] AND arrAxisCtrl[AxiseNo.AxisName.LCurlingneedleLine].Status.NoMoving
								   AND arrAxisCtrl[AxiseNo.AxisName.SCurlingneedleLine].Cmd.arrbRealPoint[1] AND arrAxisCtrl[AxiseNo.AxisName.SCurlingneedleLine].Status.NoMoving THEN
									arrAxisCtrl[AxiseNo.AxisName.LCurlingneedleWhirling].Cmd.bHome:=FALSE;//尾卷长卷针旋转回原点
									arrAxisCtrl[AxiseNo.AxisName.SCurlingneedleWhirling].Cmd.bHome:=FALSE;//尾卷短卷针旋转回原点
									TailCurlStep1:=40; 
							END_IF
			
	40:
						IF 	arrAxisCtrl[AxiseNo.AxisName.LCurlingneedleLine].Cmd.arrbRealPoint[1] AND arrAxisCtrl[AxiseNo.AxisName.LCurlingneedleLine].Status.NoMoving AND
						arrAxisCtrl[AxiseNo.AxisName.LCurlingneedleLine].Cmd.arrbRealPoint[1] AND arrAxisCtrl[AxiseNo.AxisName.LCurlingneedleLine].Status.NoMoving THEN
						//IF NOT tTailCurlTON.Q THEN
								arrAxisCtrl[AxiseNo.AxisName.LCurlingneedleWhirling].Cmd.bHome:=TRUE;//尾卷长卷针旋转回原点
								arrAxisCtrl[AxiseNo.AxisName.SCurlingneedleWhirling].Cmd.bHome:=TRUE;//尾卷短卷针旋转回原点
								//tTailCurlTON.IN:=TRUE;
						//ELSE
								//IF arrAxisCtrl[AxiseNo.AxisName.LCurlingneedleWhirling].Status.Homed AND arrAxisCtrl[AxiseNo.AxisName.LCurlingneedleWhirling].Status.NoMoving AND 
								//	arrAxisCtrl[AxiseNo.AxisName.SCurlingneedleWhirling].Status.Homed AND arrAxisCtrl[AxiseNo.AxisName.SCurlingneedleWhirling].Status.NoMoving  THEN
									//tTailCurlTON.IN:=FALSE;
									TailCurlStep1:=50; 
								//END_IF	
						END_IF
	50://
					IF arrAxisCtrl[AxiseNo.AxisName.LCurlingneedleWhirling].Status.Homed AND arrAxisCtrl[AxiseNo.AxisName.LCurlingneedleWhirling].Status.NoMoving AND 
						arrAxisCtrl[AxiseNo.AxisName.SCurlingneedleWhirling].Status.Homed AND arrAxisCtrl[AxiseNo.AxisName.SCurlingneedleWhirling].Status.NoMoving  THEN
							TailCurlStep1:=51; 	
                            tTailCurlTON.IN:=FALSE;					
					END_IF
	51://夹电芯伸缩回原
			//IF arrAxisCtrl[AxiseNo.AxisName.TailCurlLine].Status.Homed AND arrAxisCtrl[AxiseNo.AxisName.TailCurlLine].Status.NoMoving THEN
				arrAxisCtrl[AxiseNo.AxisName.TailCurlRetracting].Cmd.bHome:=TRUE;//尾卷夹电芯伸缩回原点
				TailCurlStep1:=52; 
				tTailCurlTON.IN:=TRUE;
			//END_IF
	52:
		IF arrAxisCtrl[AxiseNo.AxisName.TailCurlRetracting].Status.Homed AND arrAxisCtrl[AxiseNo.AxisName.TailCurlRetracting].Status.NoMoving AND
           tTailCurlTON.Q  THEN
			arrAxisCtrl[AxiseNo.AxisName.TailCurlRetracting].Cmd.bHome:=FALSE;
			TailCurlStep1:=53; 
			tTailCurlTON.IN:=FALSE;
		END_IF					
					
	53://夹电芯平移回原
					IF 	arrAxisCtrl[AxiseNo.AxisName.LCurlingneedleLine].Cmd.arrbRealPoint[1] AND 	arrAxisCtrl[AxiseNo.AxisName.SCurlingneedleLine].Cmd.arrbRealPoint[1] AND 			
						arrAxisCtrl[AxiseNo.AxisName.SCurlingneedleLine].Status.Homed  AND   arrAxisCtrl[AxiseNo.AxisName.LCurlingneedleLine].Status.Homed  AND
						(arrAxisCtrl[AxiseNo.AxisName.TailCurlWhirling].Status.fSetPos<=arrAxisPar[AxiseNo.AxisName.TailCurlWhirling].arrTargetPoint[1]+1 AND
						arrAxisCtrl[AxiseNo.AxisName.TailCurlWhirling].Status.fSetPos>=arrAxisPar[AxiseNo.AxisName.TailCurlWhirling].arrTargetPoint[1]-1	) OR 
						(arrAxisCtrl[AxiseNo.AxisName.TailCurlWhirling].Status.fSetPos<=arrAxisPar[AxiseNo.AxisName.TailCurlWhirling].arrTargetPoint[2]+1 AND
						arrAxisCtrl[AxiseNo.AxisName.TailCurlWhirling].Status.fSetPos>=arrAxisPar[AxiseNo.AxisName.TailCurlWhirling].arrTargetPoint[2]-1	)  THEN
							arrAxisCtrl[AxiseNo.AxisName.TailCurlLine].Cmd.bHome:=TRUE;//尾卷夹电芯平移回原点
							TailCurlTorMark:=TRUE;//尾卷夹电芯平移力矩判断标志位
							TailCurlStep1:=54; 
							tTailCurlTON.IN:=TRUE;
                     ELSE
						    TailCurlStep1:=0; 
						     Mach_Control.WJ_b.Error[8]:=TRUE;//夹电芯平移回原点时条件不满足报警
					END_IF					
	54:
		IF arrAxisCtrl[AxiseNo.AxisName.TailCurlLine].Status.Homed AND arrAxisCtrl[AxiseNo.AxisName.TailCurlLine].Status.NoMoving AND
            tTailCurlTON.Q  THEN
			arrAxisCtrl[AxiseNo.AxisName.TailCurlLine].Cmd.bHome:=FALSE;
			TailCurlStep1:=60; 	
            tTailCurlTON.IN:=FALSE;	
		END_IF		
	
	60://夹电芯平移轴移至初始位、夹电芯伸缩轴移至初始位
						IF arrAxisCtrl[AxiseNo.AxisName.TailCurlLine].Status.Homed AND arrAxisCtrl[AxiseNo.AxisName.TailCurlLine].Status.NoMoving THEN
							TailCurlTorMark:=FALSE;//尾卷夹电芯平移力矩判断标志位
							IF arrAxisCtrl[AxiseNo.AxisName.TailCurlLine].Cmd.arrbRealPoint[1] THEN
								arrAxisCtrl[AxiseNo.AxisName.TailCurlLine].Cmd.iGoSetPos:=0;
							ELSE
								arrAxisCtrl[AxiseNo.AxisName.TailCurlLine].Cmd.iGoSetPos:=1;
							END_IF
						END_IF
						IF 	arrAxisCtrl[AxiseNo.AxisName.TailCurlRetracting].Status.Homed AND arrAxisCtrl[AxiseNo.AxisName.TailCurlRetracting].Status.NoMoving THEN
							IF arrAxisCtrl[AxiseNo.AxisName.TailCurlRetracting].Cmd.arrbRealPoint[1] THEN
								arrAxisCtrl[AxiseNo.AxisName.TailCurlRetracting].Cmd.iGoSetPos:=0;
							ELSE
								arrAxisCtrl[AxiseNo.AxisName.TailCurlRetracting].Cmd.iGoSetPos:=1;
							END_IF
						END_IF	
						IF arrAxisCtrl[AxiseNo.AxisName.TailCurlLine].Cmd.arrbRealPoint[1] AND  arrAxisCtrl[AxiseNo.AxisName.TailCurlLine].Status.NoMoving AND
							arrAxisCtrl[AxiseNo.AxisName.TailCurlRetracting].Cmd.arrbRealPoint[1] AND arrAxisCtrl[AxiseNo.AxisName.TailCurlRetracting].Status.NoMoving THEN
							TailCurlStep1:=70;
						END_IF
	70:		
			IF arrAxisCtrl[AxiseNo.AxisName.TailCurlLine].Cmd.arrbRealPoint[1] AND  arrAxisCtrl[AxiseNo.AxisName.TailCurlLine].Status.NoMoving AND
			arrAxisCtrl[AxiseNo.AxisName.TailCurlRetracting].Cmd.arrbRealPoint[1] AND arrAxisCtrl[AxiseNo.AxisName.TailCurlRetracting].Status.NoMoving THEN
			//IF NOT tTailCurlTON.Q THEN
				arrAxisCtrl[AxiseNo.AxisName.TailCurlUpDown].Cmd.bHome:=TRUE;//尾卷夹电芯升降回原点
				arrAxisCtrl[AxiseNo.AxisName.TailCurlSEPTAUpDown].Cmd.bHome:=TRUE;//尾卷夹膜升降回原点
				//tTailCurlTON.IN:=TRUE;
			//ELSE
				IF NOT  arrAxisCtrl[AxiseNo.AxisName.TailCurlUpDown].Status.Homed AND NOT arrAxisCtrl[AxiseNo.AxisName.TailCurlSEPTAUpDown].Status.Homed THEN
					TailCurlStep1:=75;
				END_IF
			END_IF	
	75:
		IF arrAxisCtrl[AxiseNo.AxisName.TailCurlUpDown].Status.Homed AND arrAxisCtrl[AxiseNo.AxisName.TailCurlUpDown].Status.NoMoving AND 
			arrAxisCtrl[AxiseNo.AxisName.TailCurlSEPTAUpDown].Status.Homed AND arrAxisCtrl[AxiseNo.AxisName.TailCurlSEPTAUpDown].Status.NoMoving THEN
			arrAxisCtrl[AxiseNo.AxisName.TailCurlUpDown].Cmd.bHome:=FALSE;//尾卷夹电芯升降回原点
			arrAxisCtrl[AxiseNo.AxisName.TailCurlSEPTAUpDown].Cmd.bHome:=FALSE;//尾卷夹膜升降回原点
			TailCurlStep1:=90;
		END_IF
    (*
    80:		
	     IF  arrAxisCtrl[AxiseNo.AxisName.TailCurlLine].Status.Homed AND arrAxisCtrl[AxiseNo.AxisName.TailCurlRetracting].Status.Homed AND
			 arrAxisCtrl[AxiseNo.AxisName.TailCurlLine].Cmd.arrbRealPoint[1] AND arrAxisCtrl[AxiseNo.AxisName.TailCurlRetracting].Cmd.arrbRealPoint[1] AND
             arrAxisCtrl[AxiseNo.AxisName.TailCurlWhirling].Status.fSetPos <5 (*AND NOT  arrAxisCtrl[AxiseNo.AxisName.TailCurlWhirling].Io.biHomeSwitch*) AND
             arrAxis[AxiseNo.AxisName.TailCurlWhirling].Status.Homed THEN
			      arrAxisPar[AxiseNo.AxisName.TailCurlWhirling].arrTargetPoint[10]:=5;
					IF arrAxisCtrl[AxiseNo.AxisName.TailCurlWhirling].Cmd.arrbRealPoint[10] AND NOT   arrAxis[AxiseNo.AxisName.TailCurlWhirling].Status.NotMoving THEN
						arrAxisCtrl[AxiseNo.AxisName.TailCurlWhirling].Cmd.iGoSetPos:=0;
						TailCurlWhirlTorMark:=FALSE;//尾卷夹电芯旋转力矩判断标志位
						TailCurlStep1:=81;
					ELSE
						arrAxisCtrl[AxiseNo.AxisName.TailCurlWhirling].Cmd.iGoSetPos:=10;
						TailCurlWhirlTorMark:=TRUE;//尾卷夹电芯旋转力矩判断标志位
					END_IF
		 END_IF
		 
	81:	
       IF arrAxis[AxiseNo.AxisName.TailCurlWhirling].Status.Homed  THEN
          arrAxisCtrl[AxiseNo.AxisName.TailCurlWhirling].Cmd.bHome:=TRUE;//尾卷夹旋转回原点
		  TailCurlWhirlTorMark:=TRUE;//尾卷夹电芯旋转力矩判断标志位
		  TailCurlStep1:=82;	
	 END_IF  
		
	82:	
      IF 	arrAxisCtrl[AxiseNo.AxisName.TailCurlWhirling].Status.Homed AND arrAxis[AxiseNo.AxisName.TailCurlWhirling].Status.NotMoving THEN	
		    arrAxisCtrl[AxiseNo.AxisName.TailCurlWhirling].Cmd.bHome:=FALSE;//尾卷夹旋转回原点
		    TailCurlStep1:=90;	
		   	TailCurlWhirlTorMark:=FALSE;//尾卷夹电芯旋转力矩判断标志位
	  END_IF
	 	IF   arrAxisCtrl[AxiseNo.AxisName.TailCurlWhirling].Status.fSetPos <-10 AND NOT arrAxisCtrl[AxiseNo.AxisName.TailCurlWhirling].Io.biHomeSwitch THEN
			 arrAxisCtrl[AxiseNo.AxisName.TailCurlWhirling].Cmd.bHome:=FALSE;//尾卷夹旋转回原点
			  arrAxisCtrl[AxiseNo.AxisName.TailCurlWhirling].Cmd.bStop:=TRUE;
			  TailCurlWhirlTorMark:=FALSE;//尾卷夹电芯旋转力矩判断标志位
			  TailCurlStep1:=9999;		
		END_IF		
		*)
 
	90://夹电芯旋转轴旋转至初始位
		IF 	arrAxis[AxiseNo.AxisName.TailCurlWhirling].Status.Homed AND arrAxis[AxiseNo.AxisName.TailCurlWhirling].Status.NotMoving AND
           arrAxisCtrl[AxiseNo.AxisName.TailCurlLine].Cmd.arrbRealPoint[1] AND arrAxisCtrl[AxiseNo.AxisName.TailCurlRetracting].Cmd.arrbRealPoint[1]  THEN
			IF arrAxisCtrl[AxiseNo.AxisName.TailCurlWhirling].Cmd.arrbRealPoint[1] THEN
				arrAxisCtrl[AxiseNo.AxisName.TailCurlWhirling].Cmd.iGoSetPos:=0;
				TailCurlWhirlTorMark:=FALSE;//尾卷夹电芯旋转力矩判断标志位
				TailCurlStep1:=100;
			ELSE
				arrAxisCtrl[AxiseNo.AxisName.TailCurlWhirling].Cmd.iGoSetPos:=1;
				TailCurlWhirlTorMark:=TRUE;//尾卷夹电芯旋转力矩判断标志位
			END_IF
		END_IF
	100://各轴移至初始位
		IF 	arrAxisCtrl[AxiseNo.AxisName.LCurlingneedleWhirling].Status.Homed AND arrAxisCtrl[AxiseNo.AxisName.LCurlingneedleWhirling].Status.NoMoving THEN
			IF arrAxisCtrl[AxiseNo.AxisName.LCurlingneedleWhirling].Cmd.arrbRealPoint[1] THEN
				arrAxisCtrl[AxiseNo.AxisName.LCurlingneedleWhirling].Cmd.iGoSetPos:=0;
			ELSE
				arrAxisCtrl[AxiseNo.AxisName.LCurlingneedleWhirling].Cmd.iGoSetPos:=1;//尾卷长卷针旋转至初始位
			END_IF
		END_IF				
		IF 	arrAxisCtrl[AxiseNo.AxisName.LCurlingneedleLine].Status.Homed AND arrAxisCtrl[AxiseNo.AxisName.LCurlingneedleLine].Status.NoMoving THEN
			IF arrAxisCtrl[AxiseNo.AxisName.LCurlingneedleLine].Cmd.arrbRealPoint[1] THEN
				arrAxisCtrl[AxiseNo.AxisName.LCurlingneedleLine].Cmd.iGoSetPos:=0;
			ELSE
				arrAxisCtrl[AxiseNo.AxisName.LCurlingneedleLine].Cmd.iGoSetPos:=1;//尾卷长卷针平移至初始位
			END_IF
		END_IF		
	
		IF 	arrAxisCtrl[AxiseNo.AxisName.SCurlingneedleWhirling].Status.Homed AND arrAxisCtrl[AxiseNo.AxisName.SCurlingneedleWhirling].Status.NoMoving THEN
			IF arrAxisCtrl[AxiseNo.AxisName.SCurlingneedleWhirling].Cmd.arrbRealPoint[1] THEN
				arrAxisCtrl[AxiseNo.AxisName.SCurlingneedleWhirling].Cmd.iGoSetPos:=0;
			ELSE
				arrAxisCtrl[AxiseNo.AxisName.SCurlingneedleWhirling].Cmd.iGoSetPos:=1;//尾卷短卷针旋转至初始位
			END_IF
		END_IF				
		IF 	arrAxisCtrl[AxiseNo.AxisName.SCurlingneedleLine].Status.Homed AND arrAxisCtrl[AxiseNo.AxisName.SCurlingneedleLine].Status.NoMoving THEN
			IF arrAxisCtrl[AxiseNo.AxisName.SCurlingneedleLine].Cmd.arrbRealPoint[1] THEN
				arrAxisCtrl[AxiseNo.AxisName.SCurlingneedleLine].Cmd.iGoSetPos:=0;
			ELSE
				arrAxisCtrl[AxiseNo.AxisName.SCurlingneedleLine].Cmd.iGoSetPos:=1;//尾卷短卷针平移至初始位
			END_IF
		END_IF		
				
		IF 	arrAxisCtrl[AxiseNo.AxisName.TailCurlSEPTAUpDown].Status.Homed AND arrAxisCtrl[AxiseNo.AxisName.TailCurlSEPTAUpDown].Status.NoMoving THEN
			IF arrAxisCtrl[AxiseNo.AxisName.TailCurlSEPTAUpDown].Cmd.arrbRealPoint[1] THEN
				arrAxisCtrl[AxiseNo.AxisName.TailCurlSEPTAUpDown].Cmd.iGoSetPos:=0;
			ELSE
				arrAxisCtrl[AxiseNo.AxisName.TailCurlSEPTAUpDown].Cmd.iGoSetPos:=1;//尾卷夹膜升降到初始位
			END_IF
		END_IF
		IF 	arrAxisCtrl[AxiseNo.AxisName.TailCurlUpDown].Status.Homed AND arrAxisCtrl[AxiseNo.AxisName.TailCurlUpDown].Status.NoMoving THEN
			IF arrAxisCtrl[AxiseNo.AxisName.TailCurlUpDown].Cmd.arrbRealPoint[1] THEN
				arrAxisCtrl[AxiseNo.AxisName.TailCurlUpDown].Cmd.iGoSetPos:=0;
			ELSE
				arrAxisCtrl[AxiseNo.AxisName.TailCurlUpDown].Cmd.iGoSetPos:=1;//尾卷夹电芯升降至初始位
			END_IF
		END_IF				
		IF arrAxisCtrl[AxiseNo.AxisName.LCurlingneedleWhirling].Cmd.arrbRealPoint[1] AND arrAxisCtrl[AxiseNo.AxisName.LCurlingneedleWhirling].Status.NoMoving AND 
			arrAxisCtrl[AxiseNo.AxisName.LCurlingneedleLine].Cmd.arrbRealPoint[1] AND arrAxisCtrl[AxiseNo.AxisName.LCurlingneedleLine].Status.NoMoving AND 
			arrAxisCtrl[AxiseNo.AxisName.LCurlingneedleWhirling].Cmd.arrbRealPoint[1] AND arrAxisCtrl[AxiseNo.AxisName.LCurlingneedleWhirling].Status.NoMoving AND 
			arrAxisCtrl[AxiseNo.AxisName.LCurlingneedleLine].Cmd.arrbRealPoint[1] AND arrAxisCtrl[AxiseNo.AxisName.LCurlingneedleLine].Status.NoMoving AND 
			arrAxisCtrl[AxiseNo.AxisName.TailCurlSEPTAUpDown].Cmd.arrbRealPoint[1] AND arrAxisCtrl[AxiseNo.AxisName.TailCurlSEPTAUpDown].Status.NoMoving AND 
			arrAxisCtrl[AxiseNo.AxisName.TailCurlUpDown].Cmd.arrbRealPoint[1] AND arrAxisCtrl[AxiseNo.AxisName.TailCurlUpDown].Status.NoMoving THEN
			TailCurlStep1:=110;
		END_IF	
	110://夹膜平移回初始位
				IF arrAxisCtrl[AxiseNo.AxisName.TailCurlSEPTALine].Cmd.arrbRealPoint[1] AND arrAxis[AxiseNo.AxisName.TailCurlSEPTALine].Status.NotMoving THEN	
							TailCurlStep1:=120;
							
				ELSE
							IF  arrAxisCtrl[AxiseNo.AxisName.TailCurlLine].Status.Homed AND arrAxisCtrl[AxiseNo.AxisName.TailCurlLine].Cmd.arrbRealPoint[1]
								AND arrAxisCtrl[AxiseNo.AxisName.CaDTCarryingUpDown].Cmd.arrbRealPoint[5]
                                (*TailCurlSEPTALineGoargee OR arrAxis[AxiseNo.AxisName.TailCurlSEPTALine].NcToPlc.SetPos<= arrAxisPar[AxiseNo.AxisName.TailCurlSEPTALine].arrTargetPoint[1]+50*) THEN	
									IF 	arrAxis[AxiseNo.AxisName.TailCurlSEPTALine].Status.Homed AND arrAxis[AxiseNo.AxisName.TailCurlSEPTALine].Status.NotMoving THEN
												IF arrAxisCtrl[AxiseNo.AxisName.TailCurlSEPTALine].Cmd.arrbRealPoint[1] THEN
													arrAxisCtrl[AxiseNo.AxisName.TailCurlSEPTALine].Cmd.iGoSetPos:=0;
													TailCurlSEPTATorMark:=FALSE;//夹膜平移力矩判断标志
												ELSE
													arrAxisCtrl[AxiseNo.AxisName.TailCurlSEPTALine].Cmd.iGoSetPos:=1;//尾卷夹膜平移至初始位
													TailCurlSEPTATorMark:=TRUE;//夹膜平移力矩判断标志
												END_IF
									END_IF		
							ELSE
										tTailCurlTON.IN:=FALSE;
										Mach_Control.WJ_b.Error[2]:=TRUE;//夹膜平移回原点条件不满足报警
										Tailcurl_Gohoming:=FALSE;//尾卷回原点中
										TailCurlStep1:=9999;		
							END_IF
				END_IF
				
	120://夹电芯平移去取电芯等待位		
			 IF arrAxisCtrl[AxiseNo.AxisName.TailCurlWhirling].Cmd.arrbRealPoint[1] AND arrAxisCtrl[AxiseNo.AxisName.TailCurlUpDown].Cmd.arrbRealPoint[1] AND
				arrAxisCtrl[AxiseNo.AxisName.TailCurlSEPTALine].Cmd.arrbRealPoint[1] AND  arrAxisCtrl[AxiseNo.AxisName.TailCurlSEPTAUpDown].Cmd.arrbRealPoint[1] AND
				arrAxisCtrl[AxiseNo.AxisName.LCurlingneedleLine].Cmd.arrbRealPoint[1] AND arrAxisCtrl[AxiseNo.AxisName.SCurlingneedleLine].Cmd.arrbRealPoint[1] AND
				arrCyCtrl[arrCyNo.CylinderName.PoleSplintCy_D].Io.DIOFFSwitch AND arrCyCtrl[arrCyNo.CylinderName.TailCurlUpdownCy].Io.DIOFFSwitch AND
				 arrAxisCtrl[AxiseNo.AxisName.TailCurlLine].Status.NoMoving   AND arrAxisCtrl[AxiseNo.AxisName.TailCurlWhirling].Cmd.arrbRealPoint[1]THEN
	 
					IF arrAxisCtrl[AxiseNo.AxisName.TailCurlLine].Cmd.arrbRealPoint[11]  THEN
						arrAxisCtrl[AxiseNo.AxisName.TailCurlLine].Cmd.iGoSetPos:=0;
						WZIniti_Done:=TRUE;//负极取片回原点完成
						Tailcurl_GohomeDone:=TRUE;//尾卷回原点完成
						Tailcurl_Gohoming:=FALSE;
						TailCurlStep1:=0;
						Mach_Control.WJ_b.TailCurlStep[1]:=0;
						TailCurlStep4:=0;
						TailCurlTorMark:=FALSE;//尾卷夹电芯平移力矩判断标志位
					ELSE
						arrAxisCtrl[AxiseNo.AxisName.TailCurlLine].Cmd.iGoSetPos:=11;//夹电芯平移移至取电芯等待位
						TailCurlTorMark:=TRUE;//尾卷夹电芯平移力矩判断标志位
					END_IF	
			 END_IF		
				
	END_CASE
	
END_IF

	IF Mach_Control.U.WJ_iMode=3 AND NOT arrAxisCtrl[AxiseNo.AxisName.TailCurlWhirling].Status.Homed AND arrAxis[AxiseNo.AxisName.TailCurlWhirling].Status.Moving AND
		arrAxisCtrl[AxiseNo.AxisName.TailCurlWhirling].Status.fSetPos <-10 AND TailCurlStep1<>82 AND  arrAxis[AxiseNo.AxisName.TailCurlWhirling].Status.Homed  THEN
	    arrAxisCtrl[AxiseNo.AxisName.TailCurlWhirling].Cmd.bHome:=FALSE;//尾卷夹旋转回原点
	    arrAxisCtrl[AxiseNo.AxisName.TailCurlWhirling].Cmd.bStop:=TRUE;
	END_IF
END_ACTION

ACTION TailCurlCam:
WJ_Cam_ton[1](PT:=T#100MS);
WJ_Cam_ton[2](PT:=T#100MS);
WJ_Cam_ton[3](PT:=T#100MS);
WJ_Cam_ton[4](PT:=T#100MS);
WJ_Cam_ton[5](PT:=T#100MS);

//尾卷凸轮曲线生成
CASE  iEndWindCam  OF   
10://计算相间距
    I20:=0;
    fMaxPosEndWind:=360;         // REAL
    fMinPosEndWind:=0;          //  REAL
    iNumberOfPointEndWind:=3600; //INT
    fIntervalEndWind:=(360-0)*0.5/ iNumberOfPointEndWind ;
    bEndWindCamDataEnable:=FALSE;
   	MEMSET(ADR(arrDeltaXmm),0,SIZEOF(arrDeltaXmm)); //  ARRAY[0..3600,0..1]  OF LREAL;  
    MEMSET(ADR(arrDeltaYmm),0,SIZEOF(arrDeltaYmm)); //  ARRAY[0..3600,0..1]  OF LREAL;  
    iEndWindCam:=20;  //INT

20:
   fbRoll_New.fAngleRel:=fAngleRel:=I20*fIntervalEndWind;
   bEndWindCamDataEnable:=TRUE;
    iEndWindCam:=30;

30:
   IF NOT  bEndWindCamDataEnable      THEN
           arrDeltaXmm[I20,0] := I20;
           arrDeltaXmm[I20,1] :=fbRoll_New.AxisXmm;

           arrDeltaYmm[I20,0] :=I20;
           arrDeltaYmm[I20,1] :=fbRoll_New.AxisYmm;

         I20:=I20+1;
		IF I20>iNumberOfPointEndWind THEN

			iEndWindCam:=666;  
		ELSE
               iEndWindCam:=20;  
		 END_IF
   END_IF

END_CASE


fbRoll_New(
	Enable:=bEndWindCamDataEnable , 
    fAngleRel:=fbRoll_New.fAngleRel,
	Width:= Par.Mechaical.fCellWidth , 
	Thick:=  Par.Mechaical.fCellThick, 
	r1:=        Par.Mechaical.fCellRadii  );
fbRoll_New.AxisXmm;
fbRoll_New.AxisYmm;



fbCreatCamEndWindX(
	Reset:=                               stSysState.bReset  , 
	bCreatTable:=                     fbCreatCamEndWindX.bCreatTable  , 
	iTable:=                             TableNo.M_TailCurlLine   , 
	arrCalculateTableData:=     arrDeltaXmm , 
	axisSlave:=                         arrAxis[AxiseNo.AxisName.TailCurlSEPTALine] , 
	axisMaster:=                      arrAxis[AxiseNo.VirAxisName.VirTailCurl] , 
	bCreatTableDone=> , 
	bCreatTableError=> , 
	bError=> );
  fbCreatCamEndWindX.bCreatTableDone;
  fbCreatCamEndWindX.bCreatTableError;
  fbCreatCamEndWindX.bError;


fbCreatCamEndWindY(
	Reset:=                               stSysState.bReset  , 
	bCreatTable:=                     fbCreatCamEndWindY.bCreatTable  , 
	iTable:=                            TableNo.M_TailCurlUpDown   , 
	arrCalculateTableData:=     arrDeltaYmm , 
	axisSlave:=                        arrAxis[AxiseNo.AxisName.TailCurlSEPTAUpDown] , 
	axisMaster:=                     arrAxis[AxiseNo.VirAxisName.VirTailCurl] , 
	bCreatTableDone=> , 
	bCreatTableError=> , 
	bError=> );
  fbCreatCamEndWindY.bCreatTableDone;
  fbCreatCamEndWindY.bCreatTableError;
  fbCreatCamEndWindY.bError;
  
 tWZCreateCamTON(IN:= , PT:=T#0.5S , Q=> , ET=> );
IF Mach_Control.U.DT_iMode=3 OR Mach_Control.U.DT_iMode=0 THEN//在手动状态下
				  //从触摸屏上创建尾卷凸轮
				  rWZCreateCam_TRIG(CLK:=Mach_Control.WJ_b.CreateCamStart , Q=> );
				  IF rWZCreateCam_TRIG.Q THEN
					  tWZCreateCamTON.IN:=FALSE;
					  WZCreatCamStep0:=10;
					  Mach_Control.WJ_b.Error[0]:=FALSE;
				  END_IF
END_IF				  
				  //尾卷凸轮创建自动程序
				  CASE WZCreatCamStep0 OF
							10:
									IF NOT   tWZCreateCamTON.Q THEN
											fbCreatCamEndWindX.bCreatTable :=FALSE;
											fbCreatCamEndWindY.bCreatTable:=FALSE;
											Mach_Control.WJ_b.CreateCamDone:=FALSE;
											tWZCreateCamTON.IN:=TRUE;
									ELSE
											tWZCreateCamTON.IN:=FALSE;
											WZCreatCamStep0:=11;
									END_IF
				  
							11:
									IF  NOT WJ_Cam_ton[1].Q THEN
										arrAxisCtrl[AxiseNo.AxisName.TailCurlSEPTALine].Cmd.bStop:=TRUE;
										arrAxisCtrl[AxiseNo.AxisName.TailCurlSEPTAUpDown].Cmd.bStop:=TRUE;
										WJ_Cam_ton[1].IN:=TRUE;
									ELSE
										WJ_Cam_ton[1].IN:=FALSE;
										WZCreatCamStep0:=12;
										arrAxisCtrl[AxiseNo.AxisName.TailCurlSEPTALine].Cmd.bStop:=FALSE;
										arrAxisCtrl[AxiseNo.AxisName.TailCurlSEPTAUpDown].Cmd.bStop:=FALSE;
									END_IF
					
							12:
									IF  NOT WJ_Cam_ton[2].Q THEN
										arrAxisCtrl[AxiseNo.AxisName.TailCurlSEPTALine].Cmd.bReset:=TRUE;	
										arrAxisCtrl[AxiseNo.AxisName.TailCurlSEPTAUpDown].Cmd.bReset:=TRUE;	
										WJ_Cam_ton[2].IN:=TRUE;
									 ELSE
										 WJ_Cam_ton[2].IN:=FALSE;
										 WZCreatCamStep0:=13;
										arrAxisCtrl[AxiseNo.AxisName.TailCurlSEPTALine].Cmd.bReset:=FALSE;	
										arrAxisCtrl[AxiseNo.AxisName.TailCurlSEPTAUpDown].Cmd.bReset:=FALSE;	
									 END_IF
									
							13:
									arrAxisCtrl[AxiseNo.AxisName.TailCurlSEPTALine].Cmd.bEnable:=TRUE;
									arrAxisCtrl[AxiseNo.AxisName.TailCurlSEPTAUpDown].Cmd.bEnable:=TRUE;
									IF arrAxisCtrl[AxiseNo.AxisName.TailCurlSEPTALine].Status.Enabled AND arrAxisCtrl[AxiseNo.AxisName.TailCurlSEPTAUpDown].Status.Enabled  THEN
										 WZCreatCamStep0:=20;
									END_IF		
						
				
									
							20://计算尾卷数据
									iEndWindCam:=10;
									Mach_Control.WJ_b.CreateCamDone:=FALSE;
									WZCreatCamStep0:=30;
							30://等持凸轮数据计算完成
								IF iEndWindCam=666 THEN
									WZCreatCamStep0:=40;
								END_IF
							40://创建尾卷平移凸轮，升降凸轮
									fbCreatCamEndWindX.bCreatTable :=TRUE;
									fbCreatCamEndWindY.bCreatTable:=TRUE;
									WZCreatCamStep0:=50;
							50://等待凸轮创建完成
									IF fbCreatCamEndWindX.bCreatTableDone AND fbCreatCamEndWindY.bCreatTableDone THEN
										Mach_Control.WJ_b.CreateCamDone:=TRUE;//尾卷凸轮创建完成
										WZCreatCamStep0:=6666;
									ELSE
											IF fbCreatCamEndWindX.bCreatTableError OR fbCreatCamEndWindY.bCreatTableError THEN
												Mach_Control.WJ_b.Error[0]:=TRUE;//尾卷凸轮创建失败
												WZCreatCamStep0:=6666;
											END_IF
									END_IF
				  END_CASE
(************************************************************凸轮耦合*****************************************************************************)
//夹膜平移凸轮耦合
//fbCamInEndWindX.ParCamIn.MasterScaling:=-0.05;
fbCamInEndWindX.ParCamIn.MasterScaling:=0.05;
fbCamInEndWindX.ParCamIn.SlaveScaling:=-1;
fbCamInEndWindX(  
	Reset:=                      stSysState.bReset  , 
	bCamInExecute:=       fbCamInEndWindX.bCamInExecute, 
	iTable1:=                   TableNo.M_TailCurlLine  , 
	ParCamIn:= , 
    axisMaster:=              arrAxis[AxiseNo.VirAxisName.VirTailCurl], 
	axisSlave:=                 arrAxis[AxiseNo.AxisName.TailCurlSEPTALine]   , 
	bError=> , 
	bReady=> , 
	bInSync=> );

P2M1_MachCtrl.WJ_b.Error[1]:=fbCamInEndWindX.bError;
fbCamInEndWindX.bReady;
fbCamInEndWindX.bInSync;
//夹膜升降凸轮耦合
fbCamInEndWindY.ParCamIn.MasterScaling:=0.05;
fbCamInEndWindY(  
	Reset:=                      stSysState.bReset  , 
	bCamInExecute:=       fbCamInEndWindY.bCamInExecute, 
	iTable1:=                   TableNo.M_TailCurlUpDown  , 
	ParCamIn:=               , 
    axisMaster:=              arrAxis[AxiseNo.VirAxisName.VirTailCurl], 
	axisSlave:=                arrAxis[AxiseNo.AxisName.TailCurlSEPTAUpDown]   , 
	bError=> , 
	bReady=> , 
	bInSync=> );

P2M1_MachCtrl.WJ_b.Error[2]:=fbCamInEndWindY.bError;
fbCamInEndWindY.bReady;
fbCamInEndWindY.bInSync;
(************************************************************齿轮耦合*****************************************************************************)
tailCurl1_GearIn(
	Master:=arrAxis[AxiseNo.VirAxisName.VirTailCurl] , 
	Slave:=arrAxis[AxiseNo.AxisName.SCurlingneedleWhirling] , 
	Execute:=tailCurl1_GearIn.Execute , 
	RatioNumerator:=1 , 
	RatioDenominator:=1 , 
	Acceleration:= , 
	Deceleration:= , 
	Jerk:= , 
	BufferMode:= , 
	Options:= , 
	InGear=> , 
	Busy=> , 
	Active=> , 
	CommandAborted=> , 
	Error=> , 
	ErrorID=> );
tailCurl1_GearIn.Error;
tailCurl1_GearIn.InGear;
	
	
fTailCurl2_TRIG(CLK:=tailCurl1_GearIn.Execute  , Q=> );
tailCurl2_CamOut(
	Slave:=arrAxis[AxiseNo.AxisName.SCurlingneedleWhirling], 
	Execute:=fTailCurl2_TRIG.Q , 
	Options:= , 
	Done=> , 
	Busy=> , 
	Error=> , 
	ErrorID=> );		
	
	
	
	
tailCurl2_GearIn(
	Master:=arrAxis[AxiseNo.VirAxisName.VirTailCurl]  , 
	Slave:=arrAxis[AxiseNo.AxisName.LCurlingneedleWhirling], 
	Execute:=tailCurl2_GearIn.Execute , 
	RatioNumerator:=1 , 
	RatioDenominator:=1 , 
	Acceleration:= , 
	Deceleration:= , 
	Jerk:= , 
	BufferMode:= , 
	Options:= , 
	InGear=> , 
	Busy=> , 
	Active=> , 
	CommandAborted=> , 
	Error=> , 
	ErrorID=> );
tailCurl2_GearIn.Error;
tailCurl2_GearIn.InGear;
	
fTailCurl3_TRIG(CLK:=tailCurl2_GearIn.Execute , Q=> );
tailCurl3_CamOut(
	Slave:=arrAxis[AxiseNo.AxisName.LCurlingneedleWhirling], 
	Execute:=fTailCurl3_TRIG.Q , 
	Options:= , 
	Done=> , 
	Busy=> , 
	Error=> , 
	ErrorID=> );
END_ACTION

ACTION TorqueCheckAlarm:
//力矩超限报警断使能
	IF 	Ca_Carrying1TorMark THEN//负极搬运1平移力矩判断标志位
		 IF arrAxisCtrl[AxiseNo.AxisName.CaCarryingLine1].Status.Moving AND (ABS(Torque.Ca_Carrying1Tor)>=Torque.Ca_Carrying1TorSet)  THEN
			Torque.Ca_Carrying1TorAlarm:=TRUE;
			arrAxisCtrl[AxiseNo.AxisName.CaCarryingLine1].Cmd.bEnable:=FALSE;
			//Ca_Carrying1TorMark:=FALSE;
			//Step_InitCaDT:=0;
		END_IF
	END_IF
	IF ABS(Torque.Ca_Carrying1Tor)<Torque.Ca_Carrying1TorSet AND Sys_Control.btn.System_Rrestbtn THEN
		Torque.Ca_Carrying1TorAlarm:=FALSE;
	END_IF
	
	IF 	Ca_Carrying2TorMark THEN//负极搬运2平移力矩判断标志位
		 IF arrAxisCtrl[AxiseNo.AxisName.CaCarryingLine2].Status.Moving AND (ABS(Torque.Ca_Carrying2Tor)>=Torque.Ca_Carrying2TorSet)  THEN
			Torque.Ca_Carrying2TorAlarm:=TRUE;
			arrAxisCtrl[AxiseNo.AxisName.CaCarryingLine2].Cmd.bEnable:=FALSE;
			//Ca_Carrying2TorMark:=FALSE;
			//Step_InitCaDT:=0;
		END_IF
	END_IF
	IF ABS(Torque.Ca_Carrying2Tor)<Torque.Ca_Carrying2TorSet AND Sys_Control.btn.System_Rrestbtn THEN
		Torque.Ca_Carrying2TorAlarm:=FALSE;
	END_IF
	
	IF 	Ca_DTCarryingTorMark THEN//负极叠台搬运平移力矩判断标志位	
		 IF arrAxisCtrl[AxiseNo.AxisName.CaDTCarryingLine].Status.Moving AND (ABS(Torque.Ca_DTCarryingTor)>=Torque.Ca_DTCarryingTorSet)  THEN
			Torque.Ca_DTCarryingTorAlarm:=TRUE;
			arrAxisCtrl[AxiseNo.AxisName.CaDTCarryingLine].Cmd.bEnable:=FALSE;
			//Ca_DTCarryingTorMark:=FALSE;
			//Step_InitCaDT:=0;
		END_IF
	END_IF
	IF ABS(Torque.Ca_DTCarryingTor)<Torque.Ca_DTCarryingTorSet AND Sys_Control.btn.System_Rrestbtn THEN
		Torque.Ca_DTCarryingTorAlarm:=FALSE;
	END_IF	

//力矩超限报警断使能
	IF 	An_CarryingTorMark THEN//正极搬运1移位力矩判断标志位
		 IF arrAxisCtrl[AxiseNo.AxisName.AnCarryingLine].Status.Moving AND (ABS(Torque.An_CarryingTor)>=Torque.An_CarryingTorSet)  THEN
			Torque.An_CarryingTorAlarm:=TRUE;
			arrAxisCtrl[AxiseNo.AxisName.AnCarryingLine].Cmd.bEnable:=FALSE;
			//An_CarryingTorMark:=FALSE;//正极搬运1移位力矩判断标志位
			//Step_InitAnDT:=0;
		END_IF
	END_IF
	IF ABS(Torque.An_CarryingTor)<Torque.An_CarryingTorSet AND Sys_Control.btn.System_Rrestbtn THEN
		Torque.An_CarryingTorAlarm:=FALSE;
	END_IF
	
	IF 	An_DTCarryingTorMark THEN//正极叠台搬运力矩判断标志位	
		 IF arrAxisCtrl[AxiseNo.AxisName.AnDTCarryingLine].Status.Moving AND (ABS(Torque.An_DTCarryingTor)>=Torque.Ca_Carrying1TorSet)  THEN
			Torque.An_DTCarryingTorAlarm:=TRUE;
			arrAxisCtrl[AxiseNo.AxisName.AnDTCarryingLine].Cmd.bEnable:=FALSE;
			An_DTCarryingTorMark:=FALSE;//正极叠台搬运力矩判断标志位	
			//Step_InitAnDT:=0;
		END_IF
	END_IF
	IF ABS(Torque.An_DTCarryingTor)<Torque.Ca_Carrying1TorSet AND Sys_Control.btn.System_Rrestbtn THEN
		Torque.An_DTCarryingTorAlarm:=FALSE;
	END_IF
	
//力矩超限报警断使能
	IF 	TailCurlTorMark THEN//尾卷夹电芯平移力矩判断标志位
		 IF arrAxisCtrl[AxiseNo.AxisName.TailCurlLine].Status.Moving AND (ABS(Torque.TailCurlTor)>=Torque.TailCurlTorSet)  THEN
			Torque.TailCurlTorAlarm:=TRUE;
			arrAxisCtrl[AxiseNo.AxisName.TailCurlLine].Cmd.bEnable:=FALSE;
			//TailCurlTorMark:=FALSE;
			//TailCurlStep1:=0;
		END_IF
	END_IF
	IF ABS(Torque.TailCurlTor)<Torque.TailCurlTorSet AND Sys_Control.btn.System_Rrestbtn THEN
		Torque.TailCurlTorAlarm:=FALSE;
	END_IF
	
	IF 	TailCurlWhirlTorMark THEN//尾卷夹电芯旋转力矩判断标志位
		 IF arrAxisCtrl[AxiseNo.AxisName.TailCurlWhirling].Status.Moving AND (ABS(Torque.TailCurlWhirlTor)>=Torque.TailCurlWhirlTorSet)  THEN
			Torque.TailCurlWhirlTorAlarm:=TRUE;
			arrAxisCtrl[AxiseNo.AxisName.TailCurlWhirling].Cmd.bEnable:=FALSE;
			//TailCurlWhirlTorMark:=FALSE;
			//TailCurlStep1:=0;
		END_IF
	END_IF
	IF ABS(Torque.TailCurlWhirlTor)<Torque.TailCurlWhirlTorSet AND Sys_Control.btn.System_Rrestbtn THEN
		Torque.TailCurlWhirlTorAlarm:=FALSE;
	END_IF

	IF 	TailCurlSEPTATorMark THEN//夹膜平移力矩判断标志位
		 IF arrAxisCtrl[AxiseNo.AxisName.TailCurlSEPTALine].Status.Moving AND (ABS(Torque.TailCurlSEPTATor)>=Torque.TailCurlSEPTATorSet)  THEN
			Torque.TailCurlSEPTATorAlarm:=TRUE;
			arrAxisCtrl[AxiseNo.AxisName.TailCurlSEPTALine].Cmd.bEnable:=FALSE;
			//TailCurlSEPTATorMark:=FALSE;
			//TailCurlStep1:=0;
		END_IF
	END_IF
	IF ABS(Torque.TailCurlSEPTATor)<Torque.TailCurlSEPTATorSet AND Sys_Control.btn.System_Rrestbtn THEN
		Torque.TailCurlSEPTATorAlarm:=FALSE;
	END_IF	
(*
	IF 	TailCurlRetMark THEN//尾卷夹电芯伸缩力矩判断标志	
		 IF arrAxisCtrl[AxiseNo.AxisName.TailCurlRetracting].Status.Moving AND (ABS(Torque.TailCurlRetTor)>=Torque.TailCurlRetTorSet)  THEN
			Torque.TailCurlRetTorAlarm:=TRUE;
			arrAxisCtrl[AxiseNo.AxisName.TailCurlRetracting].Cmd.bEnable:=FALSE;
			//TailCurlRetMark:=FALSE;
			//TailCurlStep1:=0;
		END_IF
	END_IF
	IF ABS(Torque.TailCurlRetTor)<Torque.TailCurlRetTorSet AND Sys_Control.btn.System_Rrestbtn THEN
		Torque.TailCurlRetTorAlarm:=FALSE;
	END_IF	
*)
END_ACTION

ACTION Vacuum_Signal:
(**************************************************分段皮带***********************************************************)
(*
//正极模切送料分段皮带
fbAnBeltVacuum( Vacuumsel:= , 
						   	tPTtime:= , 	
							VarrCyCtrl1:=arrCyCtrl[arrCyNo.ElectValveName.AnBeltVacuum] , 
							VarrCyCtrl2:=arrCyCtrl[arrCyNo.ElectValveName.AnBeltVacuumBark] );

//负极模切送料分段皮带
fbCaMQBeltVacuum(Vacuumsel:= , 
								tPTtime:= , 
								VarrCyCtrl1:=arrCyCtrl[arrCyNo.ElectValveName.CaMQBeltVacuum] , 
								VarrCyCtrl2:=arrCyCtrl[arrCyNo.ElectValveName.CaMQBeltVacuumBark] );

//负极送片皮带末端真空
fbCaLoadUpBeltVacuum(Vacuumsel:= , 
										tPTtime:= , 
										VarrCyCtrl1:=arrCyCtrl[arrCyNo.ElectValveName.CaLoadUpBeltVacuum] , 
										VarrCyCtrl2:=arrCyCtrl[arrCyNo.ElectValveName.CaLoadUpBeltVacuumBark] );




(**************************************************叠片吸盘***********************************************************)
//正极送片搬运升降真空
fbAnCarryingVacuum(Vacuumsel:= , 
									tPTtime:= , 
									VarrCyCtrl1:=arrCyCtrl[arrCyNo.ElectValveName.AnCarryingVacuum] , 
									VarrCyCtrl2:=arrCyCtrl[arrCyNo.ElectValveName.AnCarryingVacuumBark] );

//正极叠片搬运升降真空
fbAnDTCarryingVacuum(Vacuumsel:= , 
										tPTtime:= , 
										VarrCyCtrl1:=arrCyCtrl[arrCyNo.ElectValveName.AnDTCarryingVacuum] , 
										VarrCyCtrl2:=arrCyCtrl[arrCyNo.ElectValveName.AnDTCarryingVacuumBark] );

//正极纠偏平台真空
fbAndeviationVacuum(Vacuumsel:= , 
									tPTtime:= , 
									VarrCyCtrl1:=arrCyCtrl[arrCyNo.ElectValveName.AndeviationVacuum] , 
									VarrCyCtrl2:=arrCyCtrl[arrCyNo.ElectValveName.AndeviationVacuumBark] );

									
//负极送片搬运升降1真空
fbCaCarryingVacuum1(Vacuumsel:= , 
									tPTtime:= , 
									VarrCyCtrl1:=arrCyCtrl[arrCyNo.ElectValveName.CaCarryingVacuum1], 
									VarrCyCtrl2:=arrCyCtrl[arrCyNo.ElectValveName.CaCarryingVacuumBark1] );

//负极送片搬运升降2真空
fbCaCarryingVacuum2(Vacuumsel:= , 
									tPTtime:= , 
									VarrCyCtrl1:=arrCyCtrl[arrCyNo.ElectValveName.CaCarryingVacuum2] , 
									VarrCyCtrl2:=arrCyCtrl[arrCyNo.ElectValveName.CaCarryingVacuumBark2] );
 
//负极叠片搬运升降真空
fbCaDTCarryingVacuum(Vacuumsel:= , 
										tPTtime:= , 
										VarrCyCtrl1:=arrCyCtrl[arrCyNo.ElectValveName.CaDTCarryingVacuum] , 
										VarrCyCtrl2:=arrCyCtrl[arrCyNo.ElectValveName.CaDTCarryingVacuumBark] );
 
//负极纠偏平台真空
fbCadeviationVacuum(Vacuumsel:= , 
									tPTtime:= , 
									VarrCyCtrl1:=arrCyCtrl[arrCyNo.ElectValveName.CadeviationVacuum] , 
									VarrCyCtrl2:=arrCyCtrl[arrCyNo.ElectValveName.CadeviationVacuumBark] );

*)


(***********************************正极分段皮带皮带末端真空控制*******************************************)
(*
//正极取料中,模切皮带破真空V1
IF Mach_Control.An_b.An_MainBelting THEN
	IF arrAxisCtrl[AxiseNo.AxisName.AnCarryingUpDown].Cmd.arrbRealPoint[2] THEN
		//fbAnBeltVacuum.Vacuumsel:=2;//正极模切送料分段皮带破真空开
		arrCyCtrl[arrCyNo.ElectValveName.AnBeltVacuumBark].Cmd.bON:=TRUE;//正极模切送料分段皮带破真空打开
		arrCyCtrl[arrCyNo.ElectValveName.AnBeltVacuumBark].Cmd.bOFF:=FALSE;//正极模切送料分段皮带破真空打关
	END_IF
ELSIF Mach_Control.An_b.AN_BeltDone OR Mach_Control.U.Step[0]=20 THEN //OR Mach_Control.U.DT_iMode = 1 
	arrCyCtrl[arrCyNo.ElectValveName.AnBeltVacuumBark].Cmd.bON:=FALSE;//正极模切送料分段皮带破真空打开
	arrCyCtrl[arrCyNo.ElectValveName.AnBeltVacuumBark].Cmd.bOFF:=TRUE;//正极模切送料分段皮带破真空打关
	//fbAnBeltVacuum.Vacuumsel:=1;//正极模切送料分段皮带真空打开	
END_IF	
*)	

///V2
rtVacuum2(CLK:=Mach_Control.An_b.An_MainBelting  , Q=> );
ftVacuum2(CLK:=Mach_Control.An_b.An_MainBelting    , Q=> );
IF  rtVacuum2.Q THEN//破真空
      arrCyCtrl[arrCyNo.ElectValveName.AnBeltVacuumBark].Cmd.bON:=TRUE;//正极模切送料分段皮带破真空打开
     arrCyCtrl[arrCyNo.ElectValveName.AnBeltVacuumBark].Cmd.bOFF:=FALSE;//正极模切送料分段皮带破真空打关
END_IF
IF  ftVacuum2.Q THEN//开真空
     arrCyCtrl[arrCyNo.ElectValveName.AnBeltVacuumBark].Cmd.bOFF:=TRUE;//正极模切送料分段皮带破真空打关
    arrCyCtrl[arrCyNo.ElectValveName.AnBeltVacuumBark].Cmd.bON:=FALSE;//正极模切送料分段皮带破真空打开
END_IF




(***********************************负极分段皮带皮带末端真空控制*******************************************)
(*
//负极取料中,模切皮带破真空V1
IF Mach_Control.Ca_b.Ca_MainBelting THEN
	IF arrAxisCtrl[AxiseNo.AxisName.CaCarryingUpDown1].Cmd.arrbRealPoint[1] THEN
		arrCyCtrl[arrCyNo.ElectValveName.CaMQBeltVacuumBark].Cmd.bON:=TRUE;//负极送片皮带末端真空开	
		arrCyCtrl[arrCyNo.ElectValveName.CaMQBeltVacuumBark].Cmd.bOFF:=FALSE;//负极送片皮带末端真空关	
		//fbCaMQBeltVacuum.Vacuumsel:=2;//负极模切分段皮带破真空开
	END_IF	
ELSIF Mach_Control.Ca_b.Ca_BeltDone  OR Mach_Control.U.Step[0]=20 THEN //OR Mach_Control.U.DT_iMode = 1
	arrCyCtrl[arrCyNo.ElectValveName.CaMQBeltVacuumBark].Cmd.bON:=FALSE;//负极送片皮带末端真空开	
	arrCyCtrl[arrCyNo.ElectValveName.CaMQBeltVacuumBark].Cmd.bOFF:=TRUE;//负极送片皮带末端真空关	
	//fbCaMQBeltVacuum.Vacuumsel:=1;//负极模切分段皮带真空打开
END_IF
*)

///V2
rtVacuum3(CLK:=Mach_Control.Ca_b.Ca_MainBelting  , Q=> );
ftVacuum3(CLK:=Mach_Control.Ca_b.Ca_MainBelting    , Q=> );
IF  rtVacuum3.Q THEN//破真空
		arrCyCtrl[arrCyNo.ElectValveName.CaMQBeltVacuumBark].Cmd.bON:=TRUE;//负极模切分段皮带破真空打开
		arrCyCtrl[arrCyNo.ElectValveName.CaMQBeltVacuumBark].Cmd.bOFF:=FALSE;//负极模切分段皮带破真空打关
END_IF
IF  ftVacuum3.Q THEN//开真空
		arrCyCtrl[arrCyNo.ElectValveName.CaMQBeltVacuumBark].Cmd.bOFF:=TRUE;//负极模切分段皮带破真空打关
		arrCyCtrl[arrCyNo.ElectValveName.CaMQBeltVacuumBark].Cmd.bON:=FALSE;//负极模切分段皮带破真空打开
END_IF



(*******************************************负极缓存皮带末端真空控制**************************************************)
//负极送片搬运输出取片中 打开破真空      取片搬运复位开真空此时吸盘离开皮带5mm          
(*
//负极取料中,缓存皮带破真空V1
IF NOT  Mach_Control.U.EmptyRunMode  THEN
	IF Mach_Control.Ca_b.Ca_CacheBelting THEN
		
		IF arrAxisCtrl[AxiseNo.AxisName.CaCarryingUpDown2].Cmd.arrbRealPoint[2] THEN
			arrCyCtrl[arrCyNo.ElectValveName.CaLoadUpBeltVacuumBark].Cmd.bON:=TRUE;//负极送片皮带末端真空开	
			arrCyCtrl[arrCyNo.ElectValveName.CaLoadUpBeltVacuumBark].Cmd.bOFF:=FALSE;//负极送片皮带末端真空关	
			//fbCaLoadUpBeltVacuum.Vacuumsel:=2;//负极送片皮带末端破真空开
		END_IF
	ELSIF arrAxisCtrl[AxiseNo.AxisName.CaBelt].Status.Moving  OR Mach_Control.U.Step[0]=20 THEN //OR Mach_Control.U.DT_iMode = 1
		arrCyCtrl[arrCyNo.ElectValveName.CaLoadUpBeltVacuumBark].Cmd.bON:=FALSE;//负极送片皮带末端真空开	
		arrCyCtrl[arrCyNo.ElectValveName.CaLoadUpBeltVacuumBark].Cmd.bOFF:=TRUE;//负极送片皮带末端真空关	
		//fbCaLoadUpBeltVacuum.Vacuumsel:=1;//负极送片皮带末端真空开
	END_IF
END_IF
*)

arrCyCtrl[arrCyNo.ElectValveName.CaLoadUpBeltVacuumBark].Status.OFFState;
arrCyCtrl[arrCyNo.ElectValveName.CaLoadUpBeltVacuumBark].Status.ONState;
///V2
rtVacuum1(CLK:=Mach_Control.Ca_b.Ca_CacheBelting , Q=> );
ftVacuum1(CLK:=Mach_Control.Ca_b.Ca_CacheBelting , Q=> );
	IF rtVacuum1.Q THEN
		arrCyCtrl[arrCyNo.ElectValveName.CaLoadUpBeltVacuumBark].Cmd.bOFF:=FALSE;//负极送片皮带末端真空关
		arrCyCtrl[arrCyNo.ElectValveName.CaLoadUpBeltVacuumBark].Cmd.bON:=TRUE;//负极送片皮带末端真空开
	END_IF
	IF ftVacuum1.Q THEN
		arrCyCtrl[arrCyNo.ElectValveName.CaLoadUpBeltVacuumBark].Cmd.bOFF:=TRUE;//负极送片皮带末端真空关
		arrCyCtrl[arrCyNo.ElectValveName.CaLoadUpBeltVacuumBark].Cmd.bON:=FALSE;//负极送片皮带末端真空开
	END_IF











  //  arrAxisCtrl[AxiseNo.AxisName.CaCarryingUpDown2].Status.fActPos<= arrAxisPar[AxiseNo.AxisName.CaCarryingUpDown2].arrTargetPoint[2]-5



(*
IF  Mach_Control.U.EmptyRunMode  THEN
	IF Mach_Control.Ca_b.Ca_CacheBelting AND  arrAxisCtrl[AxiseNo.AxisName.CaCarryingUpDown2].Cmd.arrbRealPoint[2] AND
		NOT arrAxisCtrl[AxiseNo.AxisName.CaBelt].Status.Moving THEN
		arrCyCtrl[arrCyNo.ElectValveName.CaLoadUpBeltVacuumBark].Cmd.bON:=TRUE;//负极送片皮带末端真空开	
		arrCyCtrl[arrCyNo.ElectValveName.CaLoadUpBeltVacuumBark].Cmd.bOFF:=FALSE;//负极送片皮带末端真空关	
		//fbCaLoadUpBeltVacuum.Vacuumsel:=2;//负极送片皮带末端破真空开
	ELSIF arrAxisCtrl[AxiseNo.AxisName.CaBelt].Status.Moving  OR Mach_Control.U.Step[0]=20 THEN
		arrCyCtrl[arrCyNo.ElectValveName.CaLoadUpBeltVacuumBark].Cmd.bON:=FALSE;//负极送片皮带末端真空开	
		arrCyCtrl[arrCyNo.ElectValveName.CaLoadUpBeltVacuumBark].Cmd.bOFF:=TRUE;//负极送片皮带末端真空关	
		//fbCaLoadUpBeltVacuum.Vacuumsel:=1;//负极送片皮带末端真空开
	END_IF
END_IF	
*)
	

(*
//正极取料中,模切皮带破真空
IF Mach_Control.An_b.An_MainBelting THEN
	IF arrAxisCtrl[AxiseNo.AxisName.AnCarryingUpDown].Cmd.arrbRealPoint[2] THEN
		fbAnBeltVacuum.Vacuumsel:=2;//正极模切送料分段皮带破真空开
	END_IF
ELSIF Mach_Control.An_b.AN_BeltDone OR Mach_Control.U.DT_iMode = 1 OR Mach_Control.U.Step[0]=20 THEN
	fbAnBeltVacuum.Vacuumsel:=1;//正极模切送料分段皮带真空打开	
END_IF		

//负极取料中,模切皮带破真空
IF Mach_Control.Ca_b.Ca_MainBelting THEN
	IF arrAxisCtrl[AxiseNo.AxisName.CaCarryingUpDown1].Cmd.arrbRealPoint[1] THEN
		fbCaMQBeltVacuum.Vacuumsel:=2;//负极模切分段皮带破真空开
	END_IF	
ELSIF Mach_Control.Ca_b.Ca_BeltDone OR Mach_Control.U.DT_iMode = 1 OR Mach_Control.U.Step[0]=20 THEN
	fbCaMQBeltVacuum.Vacuumsel:=1;//负极模切分段皮带真空打开
END_IF


	//正极取料中,控制皮带破真空
	IF Mach_Control.An_b.An_MainBelting   THEN//AND Mach_Control.An_b.An_MainBeltOK 
			arrCyCtrl[arrCyNo.ElectValveName.AnBeltVacuumBark].Cmd.bON:=TRUE;//正极模切送料分段皮带破真空打开
			arrCyCtrl[arrCyNo.ElectValveName.AnBeltVacuumBark].Cmd.bOFF:=FALSE;//正极模切送料分段皮带破真空打关
	ELSE
			arrCyCtrl[arrCyNo.ElectValveName.AnBeltVacuumBark].Cmd.bOFF:=TRUE;//正极模切送料分段皮带破真空打关
			arrCyCtrl[arrCyNo.ElectValveName.AnBeltVacuumBark].Cmd.bON:=FALSE;//正极模切送料分段皮带破真空打开
	END_IF
	//负极取料中,控制皮带破真空
	IF Mach_Control.Ca_b.Ca_MainBelting   THEN//AND Mach_Control.Ca_b.Ca_MainBeltOK 
		arrCyCtrl[arrCyNo.ElectValveName.CaMQBeltVacuumBark].Cmd.bON:=TRUE;//负极模切分段皮带破真空打开
		arrCyCtrl[arrCyNo.ElectValveName.CaMQBeltVacuumBark].Cmd.bOFF:=FALSE;//负极模切分段皮带破真空打关
	ELSE
		arrCyCtrl[arrCyNo.ElectValveName.CaMQBeltVacuumBark].Cmd.bOFF:=TRUE;//负极模切分段皮带破真空打关
		arrCyCtrl[arrCyNo.ElectValveName.CaMQBeltVacuumBark].Cmd.bON:=FALSE;//负极模切分段皮带破真空打开
	END_IF
	IF(* Mach_Control.Ca_b.Ca_CacheBelting  AND *)Mach_Control.Ca_b.Ca_CacheBeltDLOK AND arrAxisCtrl[AxiseNo.AxisName.CaBelt].Status.NoMoving THEN
		arrCyCtrl[arrCyNo.ElectValveName.CaLoadUpBeltVacuumBark].Cmd.bOFF:=FALSE;//负极送片皮带末端真空关
		arrCyCtrl[arrCyNo.ElectValveName.CaLoadUpBeltVacuumBark].Cmd.bON:=TRUE;//负极送片皮带末端真空开					
	ELSE
		arrCyCtrl[arrCyNo.ElectValveName.CaLoadUpBeltVacuumBark].Cmd.bOFF:=TRUE;//负极送片皮带末端真空关
		arrCyCtrl[arrCyNo.ElectValveName.CaLoadUpBeltVacuumBark].Cmd.bON:=FALSE;//负极送片皮带末端真空开
	END_IF
*)
END_ACTION

ACTION WJ_SingMode:
						IF Mach_Control.TJ_b.SinStepMode THEN//尾卷单步模式
							TailCurlSinStep:=TRUE;
						ELSE
							TailCurlSinStep:=FALSE;
						END_IF
END_ACTION

END_FUNCTION_BLOCK

(* stored: Version 1.1.0.1, ProductVersion 3.1.4024.12
   POU P2Program_FB: Id {ff48b66a-0f3a-49b6-9c61-bd6d30d7a232}, SpecialFunc None
   Folder 01Ca_StandbyAuto: Id {23b83efb-7dfd-4a78-b883-6e66a920a366}
   Folder 02An_StandbyAuto: Id {cd5ab33c-33e7-4b5c-8ae6-7029009be8e4}
   Folder 03DietaiAuto: Id {d691fe72-5e60-4a5b-b59f-986c068f3230}
   Folder 04TailCurl: Id {2d9db1f1-19fa-4c26-89dd-b20d2ed7b54c}
   Folder 05StickGlue: Id {29a0655a-3855-4f98-9d33-b2ed047c9bf4}
   Folder 08Init: Id {6fa67d42-18b3-4851-a9c4-3c5268a1855f}
   Folder 09Manual: Id {4145ec0d-cf08-4bcc-9adf-a26451aaf092}
   Action _01_DT_Product: Id {6d643b7b-5b40-48fa-8a21-a59030b56bac}
   Action _01DT_Auto: Id {b75b5f78-ab29-4878-8c44-46bdb967f856}
   Action _01DT_Auto2: Id {04f8d55f-4617-4a90-a831-30461344beb0}
   Action _01DT_Auto3: Id {761fff91-75cc-4d1e-985b-19f7e385a783}
   Action _01DT_Auto4: Id {dfc5d3f0-5e02-4ffe-aeff-76e924220091}
   Action _01DT_Auto5: Id {6b265681-2012-48c5-a537-2aa08a847760}
   Action _01DT_AutoSub1_CamOut: Id {bc0824c9-4f45-4ea6-91d1-e8394d1e08d2}
   Action _01Sticker_Auto: Id {1ec92b01-9bc5-461c-8275-c5e7ee907ba1}
   Action _02BlueGlue_Auto: Id {24411b71-95cd-49ad-8532-2509bc4aeaf2}
   Action _02Sticker_Auto: Id {4faef247-1ede-4f1e-bc0b-3d8232f00e6f}
   Action _02Sticker_AutoSbu1_Scan: Id {43735cac-e08f-4ec2-906b-4d2820d7ead7}
   Action _02Sticker_AutoSbu2_NG: Id {7fed9eb8-a6d2-4b8a-9fad-31d2e76ab425}
   Action _03Rectifydev_Auto: Id {25a0f6c2-d2b9-4426-bf43-1e9d04cb0311}
   Action _04Tension_Auto: Id {b03793d8-984a-4a31-8e3a-dac90b02c90b}
   Action All_GoHome: Id {e8889d8d-c288-44f7-9a22-8dfc81392818}
   Action An_Alarm: Id {7380cd5c-211c-453c-808e-b4cbf6b83b43}
   Action An_Cam: Id {4718e708-5694-4d78-8b37-071e13301154}
   Action An_Conditions: Id {db591942-a85b-4f07-82e9-699e491aec5b}
   Action An_Gohome: Id {83239e74-87c6-438f-8764-5df8d705d23f}
   Action An_OverNG: Id {011afc7e-2d04-4747-ab6c-dc606d984c7a}
   Action An_Rectifydev: Id {ccc449a1-cf6c-4267-a739-407e3c7a54c2}
   Action An_StandbyMain: Id {d6a1760a-b5d3-4ed9-8dba-4c61cfb6eab1}
   Action An_StandbyMain2: Id {822b154d-4b92-4db6-bd6e-00153bcc683b}
   Action An_StandbySub1: Id {3a9c0cf5-1edb-4c13-9eec-0da7772de3f6}
   Action An_StandbySub2: Id {82b5ceb2-fee7-4222-b0c9-b479c529cf27}
   Action An_StandbySub3: Id {b3f8ce61-0e1f-4e32-8684-f61bceb3309d}
   Action An_StandbySub4: Id {66721a2e-ac78-4b60-9608-31aead3b2059}
   Action Ca_Alarm: Id {04590461-8061-4fa9-903e-71d3ac1b6242}
   Action Ca_Cahebelt: Id {10878c62-be07-4780-92c9-96427d74dd80}
   Action Ca_Cam: Id {12873e1c-2dca-427e-9070-380ac47dfd41}
   Action Ca_Conditions: Id {214fb6d6-8b05-4f82-b976-7070d6207382}
   Action Ca_Gohome: Id {ce09218f-7459-4fbc-8b28-af9b0758f130}
   Action Ca_OverNG: Id {f84f98bb-a1b2-4ce1-97d6-8f0649da9df1}
   Action Ca_Rectifydev: Id {9ee424f1-2624-4b52-8443-1d0421d47c66}
   Action Ca_StandbyMain: Id {678a98af-09e7-4da4-a39a-ab4aa4b42a4e}
   Action Ca_StandbyMain2: Id {dcff8189-b5ea-47d4-932a-15f79ac9922b}
   Action Ca_StandbySub1: Id {4f4328f4-d662-4184-bb9d-e603c3e02d99}
   Action Ca_StandbySub2: Id {561ff454-85f5-4b95-bf0f-029c8a638310}
   Action Ca_StandbySub3: Id {fd628cbd-ef68-436e-82fb-4dc680cae540}
   Action Ca_StandbySub4: Id {79f10142-8ee5-4a97-ac00-b155c7866751}
   Action Code: Id {515ea84f-8fc1-434d-bd0b-83904bbd50b6}
   Action Dietai_Cam: Id {3aebf957-211f-422b-b84f-4824064d2ed7}
   Action Dietai_Gohome: Id {94171a4a-14f3-4f26-89fb-f24af38266ad}
   Action DT_Alarm: Id {37a313e5-b6b4-4159-a665-4e41adca7fa3}
   Action DT_Condition: Id {ea9f997b-c961-4676-911f-d81dd86084f6}
   Action DT_SingeMode: Id {e528eccb-76c4-42d3-a6f5-669d9e75e929}
   Action GMBufferCam: Id {4d8395d1-5ab8-4eee-b360-1d16eb499a9c}
   Action GMBufferLengthCalculate: Id {1a6344b7-4c43-444d-bc2f-f0f8bcd6547a}
   Action GMEmptyFold1: Id {6fc85fdc-c8d4-4ec7-8331-671ccb947980}
   Action GMEmptyFold2: Id {79a4b93e-a6bd-4eda-a045-c1487782eacb}
   Action GMEmptyFold3: Id {827ab5c4-c978-4632-9777-4039b3ab0de5}
   Action Manual: Id {e6f679c5-7ea1-4f72-9997-1be99a2c6c9f}
   Action ModeENLimk: Id {30bb4e16-9413-42fb-94da-048eb158acbb}
   Action MotionCoe_Write: Id {41020575-d472-4e13-8e98-6318d980dd67}
   Action P2_Init: Id {16af0b7d-bde0-4a33-b066-e793414cc290}
   Action Stick_Condition: Id {6d491691-6dcf-4533-adc2-8f59ccef7d7a}
   Action Sticker_Alarm: Id {d9790525-113d-4832-8d40-858be52163ca}
   Action Sticker_Gohome: Id {110b91a9-d02b-4ebc-ad1f-d9522ade4615}
   Action StickGlue_Init: Id {c93ce707-1068-46ca-8682-3307fd269806}
   Action TailCurl_Alarm: Id {17be2edf-9978-4635-a1ab-e67f4d0b0c24}
   Action TailCurl_Auto_CamOut: Id {72784fc1-8f25-447e-a06b-3872761fbeb6}
   Action TailCurl_Auto1: Id {9312de7f-505a-423f-981d-7087ffc6f00c}
   Action TailCurl_Auto2: Id {49b6b37e-6406-4c24-824b-d60494d0c243}
   Action TailCurl_Condition: Id {7a4142b8-c225-48ac-8d7f-359b5d374af4}
   Action TailCurl_Gohome: Id {d7f9db1b-58aa-4409-80d5-a4cdd578f4b1}
   Action TailCurlCam: Id {cca7155a-7700-41b7-b06f-53f8094cb4b7}
   Action TorqueCheckAlarm: Id {9368cef5-7da8-49c8-ad73-37958a5fcbe1}
   Action Vacuum_Signal: Id {ab559ec6-3f98-42f2-92ab-58cac331ad05}
   Action WJ_SingMode: Id {d0eb5e68-a938-4084-9e04-c870824da561} *)
